FUNCTION_BLOCK "GCS7_M_DPScaleMWBL_MWBS"	// FB 61
TITLE = Scale MWBL/MWBS
//  
//COPYRIGHT:    (C) 2001  BUHLER AG, CH-9240 UZWIL, SWITZERLAND
//
//PRODUCT:      GCS7
//
//TITLE:        FB 61 Machine Control:Scale MWBL/MWBS
//              (with FB40) 
//-------------------------------------------------------------------------
//
//IDENT:        AUTHOR:             DEPT:                       DATE:
//
//FB61.2.1      A. Egli             CT3                         17-Mai-2004
//              Scale.InDisableDischargeDUMP moved to last netzwerk
//              Scale not interlocked with InDisableAirlock 
//FB61.2.0      A. Egli             CT3                         17-Jun-2002
//              New Release with one block 
//FB61.1.0      A. Egli             CT3                         23-Aug-2001
//              Make new Version FB62.5.1 with DP Scales
//
//-------------------------------------------------------------------------
//
//PURPOSE:      MANUAL : see [LL.MWBxxMAN]
//
//RESTRICTIONS: S7
//              ACCU2: Pointer to dynamic datas of the machine
//              ACCU1: Pointer to parameter datas of the machine
//              >=FB26.1.0 
//
//-------------------------------------------------------------------------
//
//
AUTHOR : EA
FAMILY : GCS7LL
NAME : Ma_MWBL
VERSION : 2.1
VAR
  Ma : UDT 20610;
  Airlock : FB 12;	//Element
  LLOutlet : FB 14;	//Element
  HLInlet : FB 14;	//Element
  Scale : FB 40;	//Element
END_VAR
VAR_TEMP
  tmpFaultStop : BOOL ;
  tmpFaultSum : BOOL ;
  tmpNext : BOOL ;
  tmpNext2 : BOOL ;
  tmpEnable : BOOL ;
  tmpEmpty : BOOL ;
  tmpDisableAirlock : BOOL ;
  tmpLenDyn : INT ;
  tmpStoreAR2 : DINT ;
END_VAR
BEGIN
NETWORK
TITLE =
      L     12;
      T     #tmpLenDyn;
NETWORK
TITLE = PC Control
      NOP   0;
//=== Test Object number =====================
      L     "SYS_DirectCtrlDB".PC.ObjectNo;	//PCControl.ObjectNo
      L     #Ma.Par.ParObjectNo;	//Input ObjectNo
      <>I;
      JC    aEnd;
//=== Test OType      ========================
      L     2061;	//Input object type
      L     "SYS_DirectCtrlDB".PC.ObjectType;	//PCControl.ObjectType
      <>I;
      JC    aEnd;
//=== Test Handshake =========================
      A     "SYS_DirectCtrlDB".PC.Hsk.FExamine;	// Handshake.FExamine
      JC    aExa;
      A     "SYS_DirectCtrlDB".PC.Hsk.FDefineCmd;	// Handshake.FDefineCmd
      O     "SYS_DirectCtrlDB".PC.Hsk.FDefinePara;	// Handshake.FDefinePara
      JC    aCmd;
aIni: L     2;	// FcInit
      UC    "SYS_DirectCtrl";
      JU    aEnd;
// Write new commands from PC to Interface of group 
aCmd: A     "SYS_DirectCtrlDB".PC.Cmd1[8];	//Cmd1[8]=CmdOff
      S     #Ma.CmdOff;
      A     "SYS_DirectCtrlDB".PC.Cmd1[9];	//Cmd1[9]=CmdOn
      S     #Ma.CmdOn;
      A     "SYS_DirectCtrlDB".PC.Cmd1[10];	//Cmd1[10]=CmdNext
      S     #Ma.CmdNext;
      A     "SYS_DirectCtrlDB".PC.Cmd1[11];	//Cmd1[11]=CmdFaultReset
      S     #Ma.CmdFaultReset;
      A     "SYS_DirectCtrlDB".PC.Cmd1[13];	//Cmd1[13]=CmdManualOn
      S     #Ma.InManual;
      A     "SYS_DirectCtrlDB".PC.Cmd2[13];	//Cmd1[13]=CmdManualOff
      R     #Ma.InManual;
//[4.0]   U     PCControl.PC.Cmd1[1]; //Cmd1[1]=CmdEmptyingOn
//[4.0]   S     #Ma.InRestdischarge;
//[4.0]   U     PCControl.PC.Cmd2[1]; //Cmd2[1]=CmdEmptyingOff
//[4.0]   R     #Ma.InRestdischarge; 
      A     "SYS_DirectCtrlDB".PC.Cmd1[2];	//Cmd1[2]=CmdDisableAirlock
      S     #Ma.InDisableAirlock;
      A     "SYS_DirectCtrlDB".PC.Cmd2[2];	//Cmd2[2]=CmdEnableAirlock
      R     #Ma.InDisableAirlock;
      A     "SYS_DirectCtrlDB".PC.Cmd1[7];	//Cmd2[2]=CmdEmptying
      S     #Ma.InOutEmptyingHopperScale;
      A     "SYS_DirectCtrlDB".PC.Cmd1[4];	//Cmd1[4]=CmdNewValue
      S     #Ma.CmdNewValue;
      A     "SYS_DirectCtrlDB".PC.Cmd1[5];	//Cmd1[5]=CmdNewJob
      S     #Ma.CmdNewJob;
      AN    "SYS_DirectCtrlDB".PC.Hsk.FDefinePara;	// Handshake.FDefinePara
      JC    aIni;
      JU    aIni;
aExa: TAR2;	// Address Dynamic data
      T     "SYS_DirectCtrlDB".GC.InDynAddr;	// -->PCControl.GC.InDynAddr
      L     #tmpLenDyn;	// Length Dynamic data
      T     "SYS_DirectCtrlDB".GC.InDynLen;	// -->PCControl.GC.InDynLen
      L     0;
      T     "SYS_DirectCtrlDB".GC.InParaAddr;	// -->PCControl.GC.InParaAddr
      T     "SYS_DirectCtrlDB".GC.InParaLen;	// -->PCControl.GC.InParaLen
      L     1;	// Code FcExamine
      UC    "SYS_DirectCtrl";
      L     10;	//Revision
      T     "SYS_DirectCtrlDB".GC.Revision;
aEnd: NOP   0;
NETWORK
TITLE = Interlocking
      NOP   0;
//===Global Group Orders===
      A     "GCS7_Gr_OutManualOn";	//Gr.OutManualOn
      S     #Ma.InManual;
      A     "GCS7_Gr_OutManualOff";	//Gr.OutManualOff
      R     #Ma.InManual;
      A     #Ma.InManual;
      S     "GCS7_Gr_InManual";	//Gr.InManual
      A     #Ma.CmdNext;
      AN    #Ma.InManual;
      O     #Ma.CmdOn;
      =     #tmpNext;
      A     #Ma.InManual;
      ON    #Ma.InLocal;
      A     #Ma.InEnable;
      AN    #Ma.CmdOff;
      =     #tmpEnable;
// Continue after Empyting
      A     #Ma.CmdNewJob;
      O     #Ma.CmdOn;
      ON    #tmpEnable;
      R     #Ma.InOutEmptyingHopperScale;	//[4.0]
//---- Low level 
      A     #HLInlet.StFalse;
      O     #HLInlet.StFault;
      O     #HLInlet.StCtoTrue;
      =     #Ma.OutEmptyInlet;
      A     #Ma.OutEmptyInlet;
      AN    #Ma.InOutEmptyingHopperScale;	//[4.0]
      A     #Ma.Par.ParWithHLInlet;
      =     #tmpEmpty;
      A     #LLOutlet.StFalse;
      O     #LLOutlet.StCtoTrue;
      =     #Ma.OutEmptyOutlet;
//--- Fault----
      O     #HLInlet.StFault;
      O     #LLOutlet.StFault;
      O     #Airlock.StFault;
      O     #Scale.StFault;
      =     #tmpFaultSum;
// 
//--- Interlocking Airlock
      A     #Ma.OutEmptyOutlet;
      AN    #Ma.InOutEmptyingHopperScale;	//[4.0]
      A     #Ma.Par.ParStopAirlockByLL;
      O     #Ma.InDisableAirlock;
      =     #tmpDisableAirlock;
      AN    #tmpDisableAirlock;
      A     #tmpEnable;
      =     #Airlock.InEnableFwd;
//[4.0->] Sequence stop DUMP scale
      AN    #Ma.InManual;
      A     #Ma.InSeqStop;
      =     #Scale.InSeqStopDUMP;	//Emptying scale, but not hopper above scale
      A     #Scale.InSeqStopDUMP;
      AN    #Scale.StDosing;
      AN    #Scale.StStarting;	//[<-4.0]
      =     #Airlock.InSeqStop;
// 
      A     #Ma.StStarted;
      O     #Ma.StEmptying;
      O     #Ma.StEmptied;
      O     #Ma.StWaiting;
      AN    #Ma.InLocal;
      AN    #Ma.InManual;
      O     #tmpNext;
      S     #Airlock.CmdNext;
      =     #tmpNext2;
// 
//--- Interlocking Scale
//[2.1]      UN    #Ma.InDisableAirlock        //[4.0] Stop scale,
//[2.1]      O     #Ma.Par.ParWithLLOutlet     //[4.0]  if no HLOutlet is used
      AN    #Airlock.StFault;
      A(;
      ON    #Airlock.StStopped;
      ON    #Ma.Par.ParWithAirlock;
      ON    #Ma.InSeqStop;
      );
      A     #tmpEnable;
      =     #Scale.InEnable;
//[2.1] Scale.InDisableDischargeDUMP moved to last netzwerk
// 
      A     #Ma.InOutEmptyingHopperScale;	//[4.0]
      AN    #Scale.InManual;
      O;
      A     #Scale.InManual;
      A     #Scale.InOutRestdischargeBin;	//[4.0]
      =     #Scale.InOutRestdischargeBin;	//[4.0]
// 
      AN    #Airlock.InEnableFwd;
      O     #Airlock.StStartedFwd;
      O     #tmpDisableAirlock;
      ON    #Ma.Par.ParWithAirlock;
      A     #tmpNext2;
      S     #Scale.CmdNext;
      A     #Ma.CmdOff;
      S     #Scale.CmdOff;
//New job 
      A     #Ma.CmdNewJob;
      S     #Scale.CmdNewJob;
      A     #Ma.CmdNewValue;
      S     #Scale.CmdNewValue;
// 
//--- Local mode --
      A     #Ma.InLocal;
      AN    #Ma.InManual;
      =     #Scale.InLocal;
      =     #Airlock.InLocal;
      =     #HLInlet.InLocal;
      A     #Scale.InLocal;	//[4.0]
      O     #Ma.Par.ParHLOutletLocal;	//[4.0]
      =     #LLOutlet.InLocal;
//--- Monitoring -------------
      A     #Airlock.StStartedFwd;
      ON    #Ma.Par.ParWithAirlock;
      O     #Scale.StDosing;
      =     #LLOutlet.InMonFalse;
//--- Fault Reset -------------
      A     #Ma.CmdFaultReset;
      S     #Scale.CmdFaultReset;
      S     #Airlock.CmdFaultReset;
      S     #HLInlet.CmdFaultReset;
      S     #LLOutlet.CmdFaultReset;
//--- Stop Point -------------
      A     #Scale.OutStopPoint;
      =     #Ma.OutStopPoint;
NETWORK
TITLE = Call Scale
      CALL  #Scale;	// Call Scale
NETWORK
TITLE = Call Motor: Airlock
      AN    #Ma.Par.ParWithAirlock;
      JC    el3;
      CALL  #Airlock;
NETWORK
TITLE = Call Digital Input: HLOutlet
el3:  AN    #Ma.Par.ParWithLLOutlet;
      JC    el4;
      CALL  #LLOutlet;
NETWORK
TITLE = Call Digital Input: LLInlet
el4:  AN    #Ma.Par.ParWithHLInlet;
      JC    StJ0;
      CALL  #HLInlet;
NETWORK
TITLE = Jump to actual state
StJ0: A     #Ma.StStopped;
      JC    S0;	// ===> State
      A     #Ma.StStarted;
      JC    S2;	// ===> State
      A     #Ma.StStarting;
      JC    S1;	// ===> State
      A     #Ma.StStopping;
      JC    S3;	// ===> State
      A     #Ma.StFault;
      JC    S4;	// ===> State
      A     #Ma.StWaiting;
      JC    S5;	// ===> State
      A     #Ma.StEmptying;
      JC    S6;	// ===> State
      A     #Ma.StEmptied;
      JC    S7;	// ===> State
NETWORK
TITLE = Stopped
xxS0: S     #Ma.StStopped;	// any Transition ===> Initialisation
//=== Logic
// Condition for StFault
S0:   A     #tmpFaultSum;
      R     #Ma.StStopped;
      JC    xxS4;	//--> ST_FAULT:
// Condition for StStarting
      AN    #Airlock.StStopped;
      A     #Ma.Par.ParWithAirlock;
      ON    #Scale.StStopped;
      R     #Ma.StStopped;
      JC    xxS1;	//--> StStarting
// Condition for StWaiting
      A     #tmpNext;
      A     #tmpEnable;
      A     #tmpEmpty;
      R     #Ma.StStopped;
      JC    xxS5;	//--> StWaiting
      JU    OUT;
NETWORK
TITLE = StStarting
xxS1: S     #Ma.StStarting;	//any Transition 
//=== Logic
// Condition for StFault
S1:   A     #tmpFaultSum;
      R     #Ma.StStarting;
      JC    xxS4;	//--> StFault
// Condition for StStarted
      A     #Scale.StDosing;
      R     #Ma.StStarting;
      JC    xxS2;	//-->StStarted
// Condition for StEmptying
      A     #Scale.StEmptying;
      O     #Scale.StEmptied;
      R     #Ma.StStarting;
      JC    xxS6;	//--> StEmptying
// Condition for StStopping
      AN    #Airlock.StStartedFwd;
      O     #Airlock.InSeqStop;
      AN    #Airlock.StStarting;
      AN    #Scale.StStarting;
      AN    #Scale.InEnable;
      R     #Ma.StStarting;
      JC    xxS3;	//-->StStopping
      JU    OUT;
NETWORK
TITLE = StStarted
xxS2: S     #Ma.StStarted;	//any Transition 
//=== Logic
// Condition for StFault
S2:   A     #tmpFaultSum;
      R     #Ma.StStarted;
      JC    xxS4;	//--> StFault
// Condition for StEmptying
      A     #Scale.StEmptying;
      O     #Scale.StEmptied;
      R     #Ma.StStarted;
      JC    xxS6;	//-->StEmptying
// Condition for StWaiting
//[4.0]   U     #tmpEmpty;     
      AN    #Ma.OutEmptyOutlet;
      ON    #Ma.Par.ParWithLLOutlet;	//[4.0]
      AN    #Ma.InOutEmptyingHopperScale;	//[4.0]
      A(;	//[5.0][PE]
      AN    #Scale.StDosing;
      O     #Scale.InDisableDischargeDUMP;	//[5.0][PE]
      );	//[5.0][PE]
      R     #Ma.StStarted;
      JC    xxS5;	//-->StWaiting
// Condition for StStopping
      AN    #Scale.StDosing;
      R     #Ma.StStarted;
      JC    xxS3;	//-->StStopping
      JU    OUT;
NETWORK
TITLE = Stopping
xxS3: S     #Ma.StStopping;	//any Transition 
//=== Logic
// Condition for StFault
S3:   A     #tmpFaultSum;
      R     #Ma.StStopping;
      JC    xxS4;	//--> StFault
// Condition for StStopped
      A     #Airlock.StStopped;
      ON    #Ma.Par.ParWithAirlock;
      A     #Scale.StStopped;
      R     #Ma.StStopping;
      JC    xxS0;	//-->StStopped
// Condition for StStarting
      A     #Airlock.StStartedFwd;
      AN    #Airlock.InSeqStop;
      O     #Scale.StDosing;
      O     #Scale.InEnable;
      R     #Ma.StStopping;
      JC    xxS1;	//-->StStarting
      JU    OUT;
NETWORK
TITLE = Fault
xxS4: S     #Ma.StFault;	//any Transition 
      JU    OUT;
//=== Logic
S4:   A     #tmpFaultSum;
      JC    OUT;
//---- Transition --
      R     #Ma.StFault;
      JU    xxS3;	//-->StStopping 
NETWORK
TITLE = StWaiting
xxS5: S     #Ma.StWaiting;	//any Transition 
      JU    OUT;
//=== Logic
// Condition for StFault
S5:   A     #tmpFaultSum;
      R     #Ma.StWaiting;
      JC    xxS4;	//--> StFault
// Condition for StDosing
      A     #Scale.StDosing;
      AN    #Scale.InDisableDischargeDUMP;	//[5.0][PE]
      R     #Ma.StWaiting;
      JC    xxS2;	//-->StDosing
// Condition for StEmptying             // [4.1]
      A     #Scale.StEmptying;	// [4.1]
      A     #LLOutlet.StFalse;	// [4.1]
      R     #Ma.StWaiting;	// [4.1]
      JC    xxS6;	//-->StEmptying // [4.1]
// Condition for StEmptied              // [4.1]
      A     #Scale.StEmptied;	// [4.1]
      A     #LLOutlet.StFalse;	// [4.1]
      R     #Ma.StWaiting;	// [4.1]
      JC    xxS7;	//-->StEmptied  // [4.1]
// Condition for StStopping
      AN    #tmpEnable;
      R     #Ma.StWaiting;
      JC    xxS0;	//-->StStopping
      JU    OUT;
NETWORK
TITLE = StEmptying
xxS6: S     #Ma.StEmptying;	//any Transition 
      JU    OUT;
//=== Logic
// Condition for StFault
S6:   A     #tmpFaultSum;
      R     #Ma.StEmptying;
      JC    xxS4;	//--> StFault
// Condition for StEmptied
      A     #Scale.StEmptied;
      R     #Ma.StEmptying;
      JC    xxS7;	//-->StEmptied
// Condition for StStopping
      AN    #Scale.StEmptying;
      R     #Ma.StEmptying;
      JC    xxS3;	//-->StStopping
      JU    OUT;
NETWORK
TITLE = StEmptied
xxS7: S     #Ma.StEmptied;	//any Transition 
      JU    OUT;
//=== Logic
// Condition for StFault
S7:   A     #tmpFaultSum;
      R     #Ma.StEmptied;
      JC    xxS4;	//--> StFault
// Condition for StStarted
      A     #Scale.StDosing;
      R     #Ma.StEmptied;
      JC    xxS2;	//-->StStarted
// Condition for StStopping
      AN    #Scale.StEmptied;
      AN    #Scale.StStarting;
      R     #Ma.StEmptied;
      JC    xxS3;	//-->StStopping
      JU    OUT;
NETWORK
TITLE = State Code
// State     StCode
// ----------------------
// StFault32
// StStopped    1
// StStarting   2
// StWaiting    3
// StStarted    4
// StStopping    7
// StEmptying     9
// StEmptied        10
OUT:  A     #Ma.StStopped;
      L     1;	//Code=StStopped
      JC    Code;
      A     #Ma.StStarted;
      L     4;	//Code=StStarted
      JC    Code;
      A     #Ma.StWaiting;
      L     3;	//Code=StWaiting
      JC    Code;
      A     #Ma.StStarting;
      L     2;	//Code=StStarting
      JC    Code;
      A     #Ma.StStopping;
      L     7;	//Code=StStopping
      JC    Code;
      A     #Ma.StEmptying;
      L     9;	//Code=StEmptying
      JC    Code;
      A     #Ma.StEmptied;
      L     10;	//Code=StEmptied
      JC    Code;
      L     32;	//Code=StFault 
Code: L     #Ma.StCode;	// Old state code
      TAK;
      T     #Ma.StCode;	// Save state code
      <>I;
      L     3;
      CC    "SYS_CBitCtrl";	//Set change bit
NETWORK
TITLE = Global End
      CLR;	//---Clear all commands
      =     #Ma.CmdOn;
      =     #Ma.CmdOff;
      =     #Ma.CmdNext;
      =     #Ma.CmdFaultReset;
      =     #Ma.CmdNewValue;
      =     #Ma.CmdNewJob;
//[2.1] Scale.InDisableDischargeDUMP moved to last netzwerk
      A     #Ma.InDisableAirlock;	//[2.1] Stop scale,
      AN    #Ma.Par.ParWithLLOutlet;	//[2.1]  if no HLOutlet is used
      O(;
      A     #LLOutlet.StFault;	//[5.0][PE]
      O     #LLOutlet.StTrue;	//[5.0][PE]
      O     #LLOutlet.StCtoFalse;	//[5.0][PE]
      A     #Ma.Par.ParWithLLOutlet;	//[2.1]
      );	//[2.1]
      =     #Scale.InDisableDischargeDUMP;	//[5.0][PE]
END_FUNCTION_BLOCK

FUNCTION_BLOCK "GCS7_M_DriveCurrent"	// FB 62
TITLE = Motor with bypass flap
//  
//COPYRIGHT:    (C) 1997  BUHLER AG, CH-9240 UZWIL,  SWITZERLAND
//
//PRODUCT:      GCS7
//
//TITLE:        FB 62 Machine Control:Drive with Current
//-------------------------------------------------------------------------
//
//IDENT:        AUTHOR:             DEPT:                       DATE:
//
//FB62.1.0      A.Egli              CT3                         5-Jul-2004
//              1st Release in S7
//
//-------------------------------------------------------------------------
//
//PURPOSE:      MANUAL : see [LL.DRCUxxMAN]
//
//RESTRICTIONS: S7
//
//-------------------------------------------------------------------------
//
AUTHOR : EA
FAMILY : GCS7LL
NAME : DRCU
VERSION : 1.0
VAR
  Ma : UDT 20620;
  Mon1 : FB 14;	//Element
  Current : FB 19;	//Element [4.0]
  Motor : FB 12;	//Element
  Release : FB 11;	//Element
END_VAR
VAR_TEMP
  tmpFaultSum : BOOL ;
  tmpLocal : BOOL ;
  tmpEnable : BOOL ;
  tmpStartReq : BOOL ;
  tmpLenDyn : INT ;
  tmpEnableRelease : BOOL ;
END_VAR
BEGIN
NETWORK
TITLE =
      L     22;
      T     #tmpLenDyn;
NETWORK
TITLE = PC Control
//=== Test Object number =====================
      L     "SYS_DirectCtrlDB".PC.ObjectNo;	//PCControl.ObjectNo
      L     #Ma.Par.ParObjectNo;	//Input ObjectNo
      <>I;
      JC    aEnd;
//=== Test OType      ========================
      L     2062;	//Input object type
      L     "SYS_DirectCtrlDB".PC.ObjectType;	//PCControl.ObjectType
      <>I;
      JC    aEnd;
//=== Test Handshake =========================
      A     "SYS_DirectCtrlDB".PC.Hsk.FExamine;	// Handshake.FExamine
      JC    aExa;
      A     "SYS_DirectCtrlDB".PC.Hsk.FDefineCmd;	// Handshake.FDefineCmd
      JC    aCmd;
      A     "SYS_DirectCtrlDB".PC.Hsk.FDefinePara;	// Handshake.FDefinePara
      JC    pPar;
aIni: L     2;	// FcInit
      UC    "SYS_DirectCtrl";
      JU    aEnd;
// Write parameter 
pPar: LAR1  P#DBX 58.0;
      L     P#6.0;
      +AR1;
      L     DBW [AR1,P#4.0];
      T     #Ma.Par.ParClearingTime;
// Write new commands from PC to Interface of group 
aCmd: A     "SYS_DirectCtrlDB".PC.Cmd1[8];	//Cmd1[8]=CmdOff
      S     #Ma.CmdOff;
      A     "SYS_DirectCtrlDB".PC.Cmd1[9];	//Cmd1[9]=CmdOn
      S     #Ma.CmdOn;
      A     "SYS_DirectCtrlDB".PC.Cmd1[10];	//Cmd1[10]=CmdNext
      S     #Ma.CmdNext;
      A     "SYS_DirectCtrlDB".PC.Cmd1[11];	//Cmd1[11]=CmdFaultReset
      S     #Ma.CmdFaultReset;
      A     "SYS_DirectCtrlDB".PC.Cmd1[13];	//Cmd1[13]=CmdManualOn
      S     #Ma.InManual;
      A     "SYS_DirectCtrlDB".PC.Cmd2[13];	//Cmd2[13]=CmdManualOff
      R     #Ma.InManual;
      R     #Motor.InManual;
      R     #Release.InManual;
      JU    aIni;
aExa: TAR2;	// Address dynamic data
      T     "SYS_DirectCtrlDB".GC.InDynAddr;	// -->PCControl.GC.InDynAddr
      L     #tmpLenDyn;	// Length Dynamic data
      T     "SYS_DirectCtrlDB".GC.InDynLen;	// -->PCControl.GC.InDynLen
      L     0;
      T     "SYS_DirectCtrlDB".GC.InParaAddr;	// -->PCControl.GC.InParaAddr
      T     "SYS_DirectCtrlDB".GC.InParaLen;	// -->PCControl.GC.InParaLen
      L     1;	// Code FcExamine
      UC    "SYS_DirectCtrl";
      L     10;	//Revision
      T     "SYS_DirectCtrlDB".GC.Revision;
aEnd: NOP   0;
NETWORK
TITLE = Interlocking
//===Global Group Orders===
      A     "GCS7_Gr_OutManualOn";	//Gr.OutManualOn
      S     #Ma.InManual;
      A     "GCS7_Gr_OutManualOff";	//Gr.OutManualOff
      R     #Ma.InManual;
      A     #Ma.InManual;
      S     "GCS7_Gr_InManual";	//Gr.InManual
      A     #Ma.InLocal;
      AN    #Ma.InManual;
      =     #tmpLocal;
//--- Fault----
      A     #Current.OutFaulted;
      A     #Ma.InMonFault;
      O     #Mon1.StFault;
      O     #Motor.StFault;
      O     #Release.StFault;
      =     #tmpFaultSum;
//---Enable----
      AN    #Ma.CmdOff;
      A     #Ma.InEnable;
      =     #tmpEnable;
//--- Local mode --
      A     #tmpLocal;
      =     #Motor.InLocal;
      =     #Mon1.InLocal;
      =     #Release.InLocal;
      =     #Current.InLocal;
//--- Fault Reset -------------
      A     #Ma.CmdFaultReset;
      S     #Mon1.CmdFaultReset;
      S     #Motor.CmdFaultReset;
      S     #Release.CmdFaultReset;
      S     #Current.CmdFaultReset;
NETWORK
TITLE = Loaded
      A     #Ma.InFeeding;
      O     #Current.OutL;
      S     #Ma.OutLoaded;
      S     #Ma.OutMonitoring;
      AN    #Motor.StStartedFwd;
      R     #Ma.OutMonitoring;
NETWORK
TITLE = Interlocking Motor
//InEnableXxx
      AN    #Current.OutFaulted;
      ON    #Ma.InMonFault;
      AN    #Mon1.StFault;
      A     #Ma.InEnable;
      A(;
      A     #Ma.OutLoaded;
      ON    #Ma.InClearing;
      );
      =     #Motor.InEnableFwd;
//CmdNext
      AN    #Ma.InManual;
      A     #Ma.CmdNext;
      A     #Motor.InEnableFwd;
      O;
      A     #Ma.InManual;
      A     #Ma.CmdOn;
      S     #Motor.CmdNext;
//CmdSeqStop
      A     #Ma.InSeqStop;
      =     #Motor.InSeqStop;
NETWORK
TITLE = Interlocking Element Release
//--------------
      A     #Motor.StStartedFwd;
      A     #Ma.OutLoaded;
      A     #Ma.InReleaseOutput;
      =     #tmpEnableRelease;
      JC    erJ1;
      L     #Ma.Par.ParDelayRelease;
      T     #Ma.Par.OutDelayDosing;
      JU    erJ2;
erJ1: AN    "GCS7_Gr_OutTick200ms";
      O     #Release.InEnable;
      JC    erJ2;
      L     #Ma.Par.OutDelayDosing;
      +     -2;
      T     #Ma.Par.OutDelayDosing;
erJ2: L     #Ma.Par.OutDelayDosing;
      L     0;
      <=I;
      A     #tmpEnableRelease;
      =     #Release.InEnable;
      SET;
      S     #Release.CmdNext;
NETWORK
TITLE = Monitoring Element Mon1
      A     #Motor.StStartedFwd;
      O     #Motor.StStartedRev;
      =     #Mon1.InMonTrue;
      CLR;
      =     #Mon1.InMonFalse;
NETWORK
TITLE = Monitoring Element Current
//Set Parameter
      L     #Ma.Par.ParCurrentNom;
      T     #Current.Par.ParLimitL;
      L     100;
      L     #Ma.Par.ParLimitMin;
      -D;
      DTR;
      L     #Ma.Par.ParCurrentNom;
      DTR;
      *R;
      L     1.000000e+02;
      /R;
      RND;
      T     #Current.Par.ParLimitLL;
      L     #Ma.Par.ParLimitMax;
      L     100;
      +I;
      DTR;
      L     #Ma.Par.ParCurrentNom;
      DTR;
      *R;
      L     1.000000e+02;
      /R;
      RND;
      T     #Current.Par.ParLimitHH;
      T     #Current.Par.ParLimitH;
      SET;
      R     #Current.Par.ParLimitsPc;
      AN    #Ma.InMonFault;
      =     #Current.Par.ParWarningLL;
      =     #Current.Par.ParWarningL;
      =     #Current.Par.ParWarningH;
      =     #Current.Par.ParWarningHH;
//Monitoring
      A     #Ma.OutMonitoring;
      =     #Current.InMonLL;
      =     #Current.InMonL;
      CLR;
      =     #Current.InMonMid;
      A     #Ma.OutMonitoring;
      =     #Current.InMonH;
      =     #Current.InMonHH;
      A     #Current.OutWarning;
      O     #Current.OutFaulted;
      A     #Motor.StStartedFwd;
      AN    #Ma.InMonFault;
      =     #Ma.OutWarning;
NETWORK
TITLE = Call Digital Input: Monitor 
      AN    #Ma.Par.ParWithMon1;
      JC    Moto;
      CALL  #Mon1;
NETWORK
TITLE = Call Motor
Moto: CALL  #Motor;
NETWORK
TITLE = Call Release
      AN    #Ma.Par.ParWithRelease;
      JC    Curr;
      CALL  #Release;
NETWORK
TITLE = Call Current
Curr: CALL  #Current;
NETWORK
TITLE = Jump to actual state
      A     #Ma.StStopped;
      JC    S0;	// ===> State
      A     #Ma.StStarted;
      JC    S2;	// ===> State
      A     #Ma.StStarting;
      JC    S1;	// ===> State
      A     #Ma.StStopping;
      JC    S3;	// ===> State
      A     #Ma.StClearing;
      JC    S5;	// ===> State
      A     #Ma.StDosing;
      JC    S6;	// ===> State
      A     #Ma.StFault;
      JC    S4;	// ===> State
NETWORK
TITLE = Stopped
xxS0: S     #Ma.StStopped;
S0:   A     #tmpFaultSum;
      R     #Ma.StStopped;
      JC    xxS4;	//--> StFault
      AN    #Motor.StStopped;
      R     #Ma.StStopped;
      JC    xxS1;	//--> StStarting
      JU    OUT;
NETWORK
TITLE = Starting
xxS1: S     #Ma.StStarting;
S1:   A     #tmpFaultSum;
      R     #Ma.StStarting;
      JC    xxS4;	//--> StFault
// Condition for StStopping
      A     #Motor.StStopped;
      O     #Motor.StStopping;
      R     #Ma.StStarting;
      JC    xxS3;	//--> StStopping
// Condition for StStarted
      A(;
      O     #Motor.StStartedFwd;
      O     #Motor.StStartedRev;
      );
      R     #Ma.StStarting;
      JC    xxS2;	//--> StStarted
      JU    OUT;
NETWORK
TITLE = Started
xxS2: S     #Ma.StStarted;
S2:   A     #tmpFaultSum;
      R     #Ma.StStarted;
      JC    xxS4;	//--> StFault
// Condition for StStopping
      AN    #Motor.StStartedRev;
      AN    #Motor.StStartedFwd;
      R     #Ma.StStarted;
      JC    xxS3;	//--> StStopping
// Condition for StEnabled
      A     #Release.StStarted;
      R     #Ma.StStarted;
      JC    xxS6;	//--> StReleased
// Condition for StClearing
      A     #Ma.InClearing;
      R     #Ma.StStarted;
      JC    xxS5;	//--> StClearing
      JU    OUT;
NETWORK
TITLE = StClearing
//any Transition 
xxS5: S     #Ma.StClearing;
      L     #Ma.Par.ParClearingTime;
      T     #Ma.Par.OutClearingTime;
//=== Logic
// Condition for StFault
S5:   A     #tmpFaultSum;
      R     #Ma.StClearing;
      JC    xxS4;	//--> StFault
// Condition for StStarted
      AN    #Motor.StStartedFwd;
      AN    #Motor.StStartedRev;
      ON    #Ma.InClearing;
      R     #Ma.StClearing;
      JC    xxS2;	//--> StStarted
// Condition for StBypassed
      L     0;
      L     #Ma.Par.OutClearingTime;
      >=I;
      R     #Ma.OutLoaded;
      JC    xxS6;	//--> StBypassed
//Clearing Time
      ON    "GCS7_Gr_OutTick500ms";	//Gr.OutTick500ms
      JC    OUT;
      L     #Ma.Par.OutClearingTime;
      +     -5;
      T     #Ma.Par.OutClearingTime;
      JU    OUT;
NETWORK
TITLE = StDosing
//any Transition 
xxS6: S     #Ma.StDosing;
//=== Logic
// Condition for StFault
S6:   A     #tmpFaultSum;
      R     #Ma.StDosing;
      JC    xxS4;	//--> StFault
// Condition for StStarted
      AN    #Release.StStarted;
      R     #Ma.StDosing;
      JC    xxS2;	//--> StStarted
// Condition for StStopping
      AN    #Motor.StStartedFwd;
      AN    #Motor.StStartedRev;
      R     #Ma.StDosing;
      JC    xxS3;	//--> StStopping
// Condition for StClearing
      A     #Ma.InClearing;
      R     #Ma.StDosing;
      JC    xxS5;	//--> StClearing
      JU    OUT;
NETWORK
TITLE = Stopping
xxS3: S     #Ma.StStopping;
S3:   A     #tmpFaultSum;
      R     #Ma.StStopping;
      JC    xxS4;	//--> StFault
// Condition for StStopped
      A     #Motor.StStopped;
      R     #Ma.StStopping;
      JC    xxS0;	//--> StStopped
// Condition for StStarting
      AN    #Motor.StStopping;
      R     #Ma.StStopping;
      JC    xxS1;	//--> StStarting
      JU    OUT;
NETWORK
TITLE = Fault
xxS4: S     #Ma.StFault;
S4:   AN    #tmpFaultSum;
      R     #Ma.StFault;
      JC    xxS3;	//--> StStopping
      JU    OUT;
NETWORK
TITLE = Global End
OUT:  CLR;	//---Clear all commands
      =     #Ma.CmdOn;
      =     #Ma.CmdOff;
      =     #Ma.CmdNext;
      =     #Ma.CmdFaultReset;
NETWORK
TITLE = State Code
// 1=StStopped    11=StStopped.Warning
// 2=StStarting   12=StStarting.Warning
// 3=StStarted    13=StStarted.Warning
// 4=StDosing     15=StDosing.Warning
// 6=StClearing   16=StClearing.Warning
// 7=StStopping   17=StStopping.Warning
//32=StFault
      L     32;	// StCode=Fault
      A     #Ma.StFault;
      JC    Code;
      L     1;	// StCode=Stopped
      A     #Ma.StStopped;
      JC    Cod1;
      L     2;	// StCode=Starting
      A     #Ma.StStarting;
      JC    Cod1;
      L     3;	// StCode=Started
      A     #Ma.StStarted;
      JC    Cod1;
      L     6;	// StCode=Clearing
      A     #Ma.StClearing;
      JC    Cod1;
      L     4;	// StCode=Dosing
      A     #Ma.StDosing;
      JC    Cod1;
      L     7;	// StCode=Stopping
Cod1: AN    #Ma.OutWarning;
      JC    Code;
      +     10;
Code: L     #Ma.StCode;	// Old state code
      TAK;
      T     #Ma.StCode;	// Save state code
      <>I;
      L     3;
      CC    "SYS_CBitCtrl";	//Set change bit
END_FUNCTION_BLOCK

FUNCTION_BLOCK "GCS7_M_DFCA"	// FB 63
TITLE = Machine DFCA, DFCB, DFBB Control
//
//COPYRIGHT:    (C) 2001  BUHLER AG, CH-9240 UZWIL, SWITZERLAND
//
//PRODUCT:      GCS7
//
//TITLE:        Machine DFCA, DFCB, DFBB Control
//              (GCPROVB Revision 11)
//-------------------------------------------------------------------------
//
//IDENT:        AUTHOR:             DEPT:                       DATE:
//
//FB63.5.0      A. Egli             CT3                         26-Oct-2004
//              FB73.5.0 with B106 
//FB63.4.0      A. Egli             CT3                         08-Dez-2003
//              FB73 with A202 
//FB63.3.0      A. Egli             CT3                         17-Jun-2002
//              DFCB, DFBB 
//FB63.2.0      A. Egli             CT3                         17-Jun-2002
//              New Release with one block 
//FB63.1.1      Ph. Engler          MU664                       31-Oct-2001
//              No Press.cmdStart if InSuspend
//FB63.1.0      A. Egli             CT3                         17-Jul-2001
//              1st Release in S7
//
//-------------------------------------------------------------------------
//
//PURPOSE:      MANUAL : see [MxxMAN]
//
//RESTRICTIONS: 
//
//-------------------------------------------------------------------------
//
AUTHOR : EA
FAMILY : GCS7LL
NAME : MA_DFCA
VERSION : 5.0
VAR
  Ma : UDT 20630;
  ElRemote : FB 14;	//Input from DFCA: (DP or Dig. Input) : Freigabe Fernbetrieb
  ElRunning : FB 14;	//Input from DFCA: (DP or Dig. Input) : Betrieb, Ganze Maschine läuft
  ElSumFault : FB 14;	//Input from DFCA: (DP or Dig. Input) : Sammelalarm
  ElFireAlarm : FB 14;	//Input from DFCA: (Dig. Input      ) : Branschutzalarm
  ElPressStart : FB 11;	//Output to DFCA : (DP or Dig. Output): Start an Presse
  ElDischargerRunning : FB 11;	//*O Output to DFCA : (DP or Dig. Output): Abtransport in Betrieb
  ElDPFault : FB 14;	//                    (Internal signal  ): DP Communication fault
  DFxx : FB 73;	//Communication modul
END_VAR
VAR_TEMP
  tmpFaultStop : BOOL ;
  tmpFaultSum : BOOL ;
  tmpLocal : BOOL ;
  tmpEnable : BOOL ;
  tmpLenDyn : INT ;
END_VAR
BEGIN
NETWORK
TITLE =
      L     20;
      T     #tmpLenDyn;
NETWORK
TITLE = Call Communication DFCA
      CALL  #DFxx (
           IOByteNr                 := #Ma.Par.ParIOByteNr);
NETWORK
TITLE = PC Control
//=== Test Object number =====================
      L     "SYS_DirectCtrlDB".PC.ObjectNo;	//PCControl.ObjectNo
      L     #Ma.Par.ParObjectNo;	//Input ObjectNo
      <>I;
      JC    aEnd;
//=== Test OType      ========================
      L     2063;	//Input object type
      L     "SYS_DirectCtrlDB".PC.ObjectType;	//PCControl.ObjectType
      <>I;
      JC    aEnd;
//=== Test Handshake =========================
      A     "SYS_DirectCtrlDB".PC.Hsk.FExamine;	// Handshake.FExamine
      JC    aExa;
      A     "SYS_DirectCtrlDB".PC.Hsk.FDefineCmd;	// Handshake.FDefineCmd
      O     "SYS_DirectCtrlDB".PC.Hsk.FDefinePara;	// Handshake.FDefinePara
      JC    aCmd;
aIni: L     2;	// FcInit
      UC    "SYS_DirectCtrl";
      JU    aEnd;
// Write new commands from PC to Interface of group 
aCmd: A     "SYS_DirectCtrlDB".PC.Cmd1[5];	//Cmd1[8]=CmdNewJob
      S     #Ma.CmdOff;
      A     "SYS_DirectCtrlDB".PC.Cmd1[8];	//Cmd1[8]=CmdOff
      S     #Ma.CmdOff;
      A     "SYS_DirectCtrlDB".PC.Cmd1[9];	//Cmd1[9]=CmdOn
      S     #Ma.CmdOn;
      A     "SYS_DirectCtrlDB".PC.Cmd1[10];	//Cmd1[10]=CmdNext
      S     #Ma.CmdNext;
      A     "SYS_DirectCtrlDB".PC.Cmd1[11];	//Cmd1[11]=CmdFaultReset
      S     #Ma.CmdFaultReset;
      A     "SYS_DirectCtrlDB".PC.Cmd1[13];	//Cmd1[13]=CmdManualOn
      S     #Ma.InManual;
      A     "SYS_DirectCtrlDB".PC.Cmd2[13];	//Cmd2[13]=CmdManualOff
      R     #Ma.InManual;
      A     "SYS_DirectCtrlDB".PC.Cmd1[6];	//Cmd1[6]=InOutCoolerOnMan.On
      S     #Ma.InOutCoolerOnMan;
      A     "SYS_DirectCtrlDB".PC.Cmd2[6];	//Cmd2[6]=Ma.InOutCoolerOnMan.Off
      R     #Ma.InOutCoolerOnMan;
      A     "SYS_DirectCtrlDB".PC.Cmd1[7];	//Cmd1[6]=Ma.InOutHeaterOnMan.On
      S     #Ma.InOutHeaterOnMan;
      A     "SYS_DirectCtrlDB".PC.Cmd2[7];	//Cmd2[6]=Ma.InOutHeaterOnMan.Off
      R     #Ma.InOutHeaterOnMan;
      A     "SYS_DirectCtrlDB".PC.Cmd1[4];	//Cmd1[6]=InOutFanOnMan.On    //[3.0]
      S     #Ma.InOutFanOnMan;
      A     "SYS_DirectCtrlDB".PC.Cmd2[4];	//Cmd2[6]=Ma.InOutFanOnMan.Off   //[3.0]
      R     #Ma.InOutFanOnMan;
      JU    aIni;
aExa: TAR2;	// Address Dynamic datas
      T     "SYS_DirectCtrlDB".GC.InDynAddr;	// -->PCControl.GC.InDynAddr
      L     #tmpLenDyn;	// Length Dynamic datas
      T     "SYS_DirectCtrlDB".GC.InDynLen;	// -->PCControl.GC.InDynLen
      L     0;
      T     "SYS_DirectCtrlDB".GC.InParaAddr;	// -->PCControl.GC.InParaAddr
      T     "SYS_DirectCtrlDB".GC.InParaLen;	// -->PCControl.GC.InParaLen
      L     1;	// Code FcExamine
      UC    "SYS_DirectCtrl";
      L     11;	//Revision
      T     "SYS_DirectCtrlDB".GC.Revision;
aEnd: NOP   0;
NETWORK
TITLE = Interlocking
//===Global Group Orders===
      A     "GCS7_Gr_OutManualOn";	//Gr.OutManualOn
      S     #Ma.InManual;
      A     "GCS7_Gr_OutManualOff";	//Gr.OutManualOff
      R     #Ma.InManual;
      A     #Ma.InManual;
      S     "GCS7_Gr_InManual";	//Gr.InManual
//--- Local mode --
      A     #Ma.InLocal;
      AN    #Ma.InManual;
      =     #tmpLocal;
      A     #tmpLocal;
      =     #ElRemote.InLocal;
      =     #ElRunning.InLocal;
      =     #ElSumFault.InLocal;
      =     #ElFireAlarm.InLocal;
      CLR;
      =     #ElPressStart.InLocal;
      =     #ElDischargerRunning.InLocal;
      A     #tmpLocal;
      ON    #Ma.Par.ParDP;
      =     #ElDPFault.InLocal;
//--- Monitoring
      A     #Ma.InRemoteMode;
      =     #ElRemote.InMonTrue;
      SET;
      =     #ElSumFault.InMonTrue;
      SET;
      =     #ElFireAlarm.InMonTrue;
      A     #Ma.Par.ParDP;
      =     #ElDPFault.InMonTrue;
//--- Fault Reset -------------
      A     #Ma.CmdFaultReset;
      S     #ElRemote.CmdFaultReset;
      S     #ElRunning.CmdFaultReset;
      S     #ElPressStart.CmdFaultReset;
      S     #ElDischargerRunning.CmdFaultReset;
      S     #ElDPFault.CmdFaultReset;
      S     #DFxx.InCommand.CmdFaultResetAll;
      AN    #Ma.CmdFaultReset;
      JC    FRJ1;
      L     #Ma.Par.ParFaultResetTime;
      T     #Ma.Par.OutFaultResetTime;
FRJ1: L     #Ma.Par.OutFaultResetTime;
      L     0;
      <=I;
      ON    "GCS7_Gr_OutTick200ms";
      JC    FRJ2;
      L     #Ma.Par.OutFaultResetTime;
      -I;
      T     #Ma.Par.OutFaultResetTime;
      L     0;
      >I;
      JC    FRJ2;
      S     #ElSumFault.CmdFaultReset;
      S     #ElFireAlarm.CmdFaultReset;
FRJ2: NOP   0;
//=============================================
//ElPressStart: Start/Stop
//=============================================
      A     #Ma.Par.ParManual;
      A     #Ma.InManual;
      O     #Ma.InEnable;
      AN    #Ma.CmdOff;
      =     #tmpEnable;
      A     #Ma.InManual;
      A     #Ma.CmdOn;
      A     #tmpEnable;
      O;
      AN    #Ma.InManual;
      A     #Ma.CmdNext;
      A     #tmpEnable;
      S     #ElPressStart.InEnable;
      S     #ElPressStart.CmdNext;
      AN    #tmpEnable;
      O     #Ma.CmdOff;
      R     #ElPressStart.InEnable;
//=============================================
//ElDischargerRunning
//=============================================
      A     #Ma.InDischargerRunning;
      =     #ElDischargerRunning.InEnable;
      S     #ElDischargerRunning.CmdNext;
NETWORK
TITLE = Commands to DFCA
      A     #ElPressStart.InEnable;
      AN    #Ma.InSuspend;	//[PE]
      =     #DFxx.InCommand.StartPress;
//------------------------------
      AN    #ElPressStart.InEnable;
      =     #DFxx.InCommand.StopPress;
//------------------------------
      A     #Ma.InDischargerRunning;
      =     #DFxx.InCommand.DischargerRunning;
//------------------------------
      A     #Ma.InOutCoolerOnMan;
      =     #DFxx.InCommand.CoolerOnMan;
//------------------------------
      A     #Ma.InOutHeaterOnMan;
      =     #DFxx.InCommand.HeaterOnMan;
//------------------------------
      A     #Ma.InOverrideLLHopper;
      =     #DFxx.InCommand.OverwriteLLHopper;
//------------------------------
      A     #Ma.InSuspend;
      =     #DFxx.InCommand.Suspend;
//------------------------------
      A     #Ma.InOutFanOnMan;	//[3.0]
      =     #DFxx.InCommand.FanOnMan;	//[3.0]
//------------------------------
      A     #Ma.CmdNewJob;
      S     #DFxx.InCommand.CmdResetTotal;
      S     #DFxx.InCommand.CmdResetTotalLiquid1;	//[3.0]
      S     #DFxx.InCommand.CmdResetTotalLiquid2;	//[3.0]
      R     #Ma.CmdNewJob;
//------------------------------
      A     #Ma.CmdResetHorn;
      S     #DFxx.InCommand.CmdResetHorn;
//------------------------------
      CLR;
      S     #DFxx.InCommand.CmdFaultResetSingle;
//------------------------------
      A     #Ma.CmdFaultReset;
      S     #DFxx.InCommand.CmdFaultResetAll;
//------------------------------
      A     #Ma.CmdSendB101;
      R     #Ma.CmdSendB101;
      S     #DFxx.In.CmdSendB101;
//------------------------------
      A     #Ma.CmdSendB102;
      R     #Ma.CmdSendB102;
      S     #DFxx.In.CmdSendB102;
//------------------------------
      A     #Ma.CmdSendB103;
      R     #Ma.CmdSendB103;
      S     #DFxx.In.CmdSendB103;
//------------------------------
      A     #Ma.CmdSendB104;
      R     #Ma.CmdSendB104;
      S     #DFxx.In.CmdSendB104;
NETWORK
TITLE = Digital outputs to DFCA
      A     #Ma.InpLL;
      =     #Ma.OutpLL;
      A     #Ma.InpLevelMiddle;
      =     #Ma.OutpLevelMiddle;
NETWORK
TITLE = Input signal from DP modul
      AN    #Ma.Par.ParDP;
      JC    IPJ0;
//===================================
      L     #DFxx.OutA101Ac.Mode;
      L     1;
      ==I;
      =     #ElRemote.InpTrue;
//===================================
      L     #DFxx.OutA101Ac.State;
      L     4;
      ==I;
      =     #ElRunning.InpTrue;
//===================================
      AN    #DFxx.OutA104Ac.SumAlarm;
      =     #ElSumFault.InpTrue;
IPJ0: NOP   0;
NETWORK
TITLE = Call Digital Input: ElRemote
      CALL  #ElRemote;
NETWORK
TITLE = Call Digital Input: ElRunning
      CALL  #ElRunning;
NETWORK
TITLE = Call Digital Input: ElSumFault
      CALL  #ElSumFault;
NETWORK
TITLE = Call Digital Input: ElFireAlarm
      CALL  #ElFireAlarm;
NETWORK
TITLE = Call ElPressStart
      CALL  #ElPressStart;
NETWORK
TITLE = Call ElDischargerRunning
      CALL  #ElDischargerRunning;
NETWORK
TITLE = Call Digital Input: ElDPFault
      ON    #Ma.Par.ParDP;
      ON    #DFxx.Out.DPFault;
      =     #ElDPFault.InpTrue;
      CALL  #ElDPFault;
NETWORK
TITLE = State
//-Relais contro:
// State:
// -Idle
// -Startup
// -Operation
// -Shutdown
//
      A     #ElRemote.StFault;
      O     #ElRunning.StFault;
      O     #ElSumFault.StFault;
      O     #ElFireAlarm.StFault;
      O     #ElPressStart.StFault;
      O     #ElDischargerRunning.StFault;
      O     #ElDPFault.StFault;
      =     #tmpFaultSum;
//=================================
//State StFault
//=================================
      A     #tmpFaultSum;
      =     #Ma.StFault;
//=================================
//State StIdle
//=================================
      L     #DFxx.OutA101Ac.State;
      L     0;
      ==I;
      A     #Ma.Par.ParDP;
      AN    #tmpFaultSum;
      O(;
      ON    #Ma.InpLL;
      ON    #Ma.InDischargerRunning;
      ON    #ElPressStart.StStarted;
      ON    #ElRemote.InpTrue;
      AN    #ElRunning.InpTrue;
      AN    #Ma.Par.ParDP;
      );
      =     #Ma.StIdle;
//=================================
//State StStartup
//=================================
      L     #DFxx.OutA101Ac.State;
      L     1;
      ==I;
      A     #Ma.Par.ParDP;
      AN    #tmpFaultSum;
      O(;
      AN    #Ma.StIdle;
      AN    #ElRunning.InpTrue;
      AN    #Ma.StFault;
      AN    #Ma.Par.ParDP;
      );
      =     #Ma.StStartup;
//=================================
//State StReady
//=================================
      L     #DFxx.OutA101Ac.State;
      L     2;
      ==I;
      A     #Ma.Par.ParDP;
      AN    #tmpFaultSum;
      =     #Ma.StReady;
//=================================
//State StFeedStartup
//=================================
      L     #DFxx.OutA101Ac.State;
      L     3;
      ==I;
      A     #Ma.Par.ParDP;
      AN    #tmpFaultSum;
      =     #Ma.StFeedStartup;
//=================================
//State StOperation
//=================================
      L     #DFxx.OutA101Ac.State;
      L     4;
      ==I;
      A     #Ma.Par.ParDP;
      AN    #tmpFaultSum;
      O(;
      AN    #Ma.Par.ParDP;
      A     #ElRunning.InpTrue;
      AN    #Ma.StIdle;
      AN    #Ma.StStartup;
      AN    #Ma.StFault;
      );
      =     #Ma.StOperation;
//=================================
//State StShutdown
//=================================
      L     #DFxx.OutA101Ac.State;
      L     5;
      ==I;
      A     #Ma.Par.ParDP;
      AN    #tmpFaultSum;
      O(;
      AN    #Ma.Par.ParDP;
      AN    #Ma.StIdle;
      AN    #Ma.StStartup;
      AN    #Ma.StFault;
      AN    #Ma.StOperation;
      );
      =     #Ma.StShutdown;
NETWORK
TITLE = Global End
      CLR;	//---Clear all commands
      =     #Ma.CmdOn;
      =     #Ma.CmdOff;
      =     #Ma.CmdNext;
      =     #Ma.CmdFaultReset;
      =     #Ma.CmdResetHorn;
NETWORK
TITLE = Digital outputs Lamp
//-----------------------------
      A     #ElRunning.InpTrue;
      =     #Ma.OutpLampRunning;
//-----------------------------
      AN    #ElSumFault.InpTrue;
      =     #Ma.OutpLampFault;
//-----------------------------
      AN    #ElFireAlarm.InpTrue;
      =     #Ma.OutpLampFireAlarm;
NETWORK
TITLE = State Code
// Same as motor
      A     #Ma.StIdle;
      L     1;	//  StCode 1=StIdle
      JC    Code;
      A     #Ma.StStartup;
      L     2;	//  StCode 2=StStartup
      JC    Code;
      A     #Ma.StReady;
      L     3;	//  StCode 3=StReady
      JC    Code;
      A     #Ma.StFeedStartup;
      L     4;	//  StCode 4=StFeedStartup
      JC    Code;
      A     #Ma.StOperation;
      L     5;	//  StCode 5=StOperation
      JC    Code;
      A     #Ma.StShutdown;
      L     6;	//  StCode 6=StShutdown
      JC    Code;
      L     32;	// StCode=Fault
Code: L     #Ma.StCode;	// Old state code
      TAK;
      T     #Ma.StCode;	// Save state code
      <>I;
      L     3;
      CC    "SYS_CBitCtrl";	//Set change bit
END_FUNCTION_BLOCK

FUNCTION_BLOCK "GCS7_M_MYFB"	// FB 64
TITLE = Machine MYEB Moisture Control
//  
//COPYRIGHT:    (C) 1997  BUHLER AG, CH-9240 UZWIL, SWITZERLAND
//
//PRODUCT:      GCS7
//
//TITLE:        Machine MYEB Moisture Control
//
//-------------------------------------------------------------------------
//
//IDENT:        AUTHOR:             DEPT:                      DATE:
//
//FB64.4.2      A. Egli             CT3                        02-Jul-2004
//              Run delay time water also when MOZ_DosingEnable is StStopped
//FB64.4.1      A. Egli             CT3                        24-Jun-2004
//              InDisableConveyor
//              FB64.3.3 GCS90S7 : InLocalWaterControl 
//FB64.4.0      A. Egli             CT3                        17-Jun-2002
//              New Release with one block 
//FB64.3.2      Ph. Engler          MU664                      19-Feb-2002
//              _Product flowmonitor: CmdRunTimeoutTime integrated
//FB64.3.1      A.Egli              CT3                        30-Oct-2001
//              InDisableWater
//FB64.3.0      S. Kalberer         CT3                        11-Oct-1999
//              Local data reduced
//FB64.2B       S. Kalberer         CT3                        10-Aug-1998
//              Clear CmdNewValue/CmdNewJob adjusted
//FB64.2A       A. Egli             CT3                        04-Mai-1998
//              StFault = StCode 32
//FB64.1A       S. Kalberer         AEE61                      22-Oct-1997
//              1st Release in S7
//
//-------------------------------------------------------------------------
//
//PURPOSE:      MANUAL : see [LL.MYBxxMAN]
//
//RESTRICTIONS: S7
//              ACCU2: Pointer to dynamic datas of the element
//              ACCU1: Pointer to parameter datas of the element
//
//-------------------------------------------------------------------------
//
AUTHOR : EA
FAMILY : GCS7LL
NAME : MYEB_Ma
VERSION : 4.2
VAR
  Ma : UDT 20640;
  MYEB_LC : FB 23;	//Element
  MYEB_GroupAlarm : FB 14;	//Element
  MYF_Product : FB 14;	//Element
  MYF_ConveyorEnable : FB 11;	//Element
  MOZ_DosingEnable : FB 11;	//Element
  MOZ_WaterValve : FB 11;	//Element
  MOZ_Product : FB 14;	//Element
  MOZ_Motor : FB 12;	//Element
END_VAR
VAR_TEMP
  tmpLenDyn : DINT ;
  tmpFaultSum : BOOL ;
  tmpFaultReset : BOOL ;
END_VAR
BEGIN
NETWORK
TITLE =
      L     30;
      T     #tmpLenDyn;	//--> Len dynamic data in byte
NETWORK
TITLE = PC Control
//=== Test Object number =====================
      L     "SYS_DirectCtrlDB".PC.ObjectNo;	//PCControl.ObjectNo
      L     #Ma.Par.ParObjectNo;	//Input ObjectNo
      <>I;
      JC    aEnd;
//=== Test OType      ========================
      L     2064;	//Input object type
      L     "SYS_DirectCtrlDB".PC.ObjectType;	//PCControl.ObjectType
      <>I;
      JC    aEnd;
//=== Test Handshake =========================
      A     "SYS_DirectCtrlDB".PC.Hsk.FExamine;	// Handshake.FExamine
      JC    aExa;
      A     "SYS_DirectCtrlDB".PC.Hsk.FDefineCmd;	// Handshake.FDefineCmd
      JC    aCmd;
      A     "SYS_DirectCtrlDB".PC.Hsk.FDefinePara;	// Handshake.FDefinePara
      JC    pPar;
aIni: L     2;	// FcInit
      UC    "SYS_DirectCtrl";
      JU    aEnd;
// Write parameter 
pPar: LAR1  P#DBX 58.0;
      L     P#6.0;
      +AR1;
      L     DBW [AR1,P#4.0];
      T     #Ma.Par.ParStartValuePc;
      L     DBW [AR1,P#6.0];
      T     #Ma.Par.ParStartValue;
      L     DBW [AR1,P#8.0];
      T     #Ma.Par.ParOffDelayFeed;
      L     DBW [AR1,P#10.0];
      T     #Ma.Par.ParOnDelayWater;
// Write new commands from PC to Interface of group 
aCmd: A     "SYS_DirectCtrlDB".PC.Cmd1[4];	//Cmd1[4]=CmdNewValue
      S     #Ma.CmdNewValue;
      A     "SYS_DirectCtrlDB".PC.Cmd1[5];	//Cmd1[5]=CmdNewJob
      S     #Ma.CmdNewJob;
      A     "SYS_DirectCtrlDB".PC.Cmd1[8];	//Cmd1[8]=CmdOff
      S     #Ma.CmdOff;
      A     "SYS_DirectCtrlDB".PC.Cmd1[9];	//Cmd1[9]=CmdOn
      S     #Ma.CmdOn;
      A     "SYS_DirectCtrlDB".PC.Cmd1[10];	//Cmd1[10]=CmdNext
      S     #Ma.CmdNext;
      A     "SYS_DirectCtrlDB".PC.Cmd1[11];	//Cmd1[11]=CmdFaultReset
      S     #Ma.CmdFaultReset;
      A     "SYS_DirectCtrlDB".PC.Cmd1[13];	//Cmd1[13]=CmdManualOn
      S     #Ma.InManual;
      A     "SYS_DirectCtrlDB".PC.Cmd1[15];	//Cmd1[15]=CmdManualWaterOn
      S     #Ma.InManualWaterControl;
      A     "SYS_DirectCtrlDB".PC.Cmd2[13];	//Cmd2[13]=CmdManualOff
      R     #Ma.InManual;
      A     "SYS_DirectCtrlDB".PC.Cmd2[15];	//Cmd2[15]=CmdManualWaterOff
      R     #Ma.InManualWaterControl;
      JU    aIni;
aExa: TAR2;	// Address Dynamic datas
      T     "SYS_DirectCtrlDB".GC.InDynAddr;	// -->PCControl.GC.InDynAddr
      L     #tmpLenDyn;	// Length Dynamic datas
      T     "SYS_DirectCtrlDB".GC.InDynLen;	// -->PCControl.GC.InDynLen
      L     0;
      T     "SYS_DirectCtrlDB".GC.InParaAddr;	// -->PCControl.GC.InParaAddr
      T     "SYS_DirectCtrlDB".GC.InParaLen;	// -->PCControl.GC.InParaLen
      L     1;	// Code FcExamine
      UC    "SYS_DirectCtrl";
      L     10;	//Revision
      T     "SYS_DirectCtrlDB".GC.Revision;
aEnd: NOP   0;
NETWORK
TITLE =  Timer switch off feed and switch on water
//Timer switch off delay feed
      A     #MOZ_WaterValve.StStarted;
      AN    #Ma.OutMoistureStart;
      A     #Ma.OutFeedReady;
      AN    #Ma.InProductFeed;
      JC    TiF0;
      R     #Ma.OutOffDelayFeedRun;
      L     0;	//Reset timervalue to zero
      T     #Ma.Par.OutOffDelayFeed;
      JU    TiW;
TiF0: A     #Ma.OutOffDelayFeedDone;
      JC    TiW;
      A     #Ma.OutOffDelayFeedRun;
      JC    TiF1;
      S     #Ma.OutOffDelayFeedRun;
      L     #Ma.Par.ParOffDelayFeed;
      T     #Ma.Par.OutOffDelayFeed;
TiF1: AN    "GCS7_Gr_OutTick1s";	//Gr.OutTick1S
      L     #Ma.Par.OutOffDelayFeed;
      JC    TiF2;
      +     -10;
      T     #Ma.Par.OutOffDelayFeed;
TiF2: L     0;
      <=I;
      R     #Ma.OutOffDelayFeedRun;
      S     #Ma.OutOffDelayFeedDone;
TiW:  A     #MOZ_Product.StTrue;
      O     #MOZ_Product.StCtoTrue;
      A(;	//[4.2]
      A     #MOZ_WaterValve.StStopped;
      O     #MOZ_DosingEnable.StStopped;	//[4.2]
      );	//[4.2]
      A     #Ma.OutFeedReady;
      A     #Ma.InProductFeed;
      JC    TiW0;
      R     #Ma.OutOnDelayWaterRun;
      L     0;	//Reset timervalue to zero
      T     #Ma.Par.OutOnDelayWater;
      JU    TiE;
//Timer swtich on delay water
TiW0: A     #Ma.OutOnDelayWaterDone;
      JC    TiE;
      A     #Ma.OutOnDelayWaterRun;
      JC    TiW1;
      S     #Ma.OutOnDelayWaterRun;
      L     #Ma.Par.ParOnDelayWater;
      T     #Ma.Par.OutOnDelayWater;
TiW1: AN    "GCS7_Gr_OutTick1s";	//Gr.OutTick1S
      L     #Ma.Par.OutOnDelayWater;
      JC    TiW2;
      +     -10;
      T     #Ma.Par.OutOnDelayWater;
TiW2: L     0;
      <=I;
      R     #Ma.OutOnDelayWaterRun;
      S     #Ma.OutOnDelayWaterDone;
//---Reset timer Done bit
TiE:  AN    #Ma.InProductFeed;
      O     #MOZ_Product.StFalse;
      R     #Ma.OutOnDelayWaterDone;
      A     #Ma.InProductFeed;
      R     #Ma.OutOffDelayFeedDone;
NETWORK
TITLE =  Set moisture StartValue or StartValuePc [%]
      A     #Ma.InManualWaterControl;
      O     #Ma.InLocalWaterControl;	//[3.3] InLocalWaterControl
      O     #Ma.StStopped;
      ON    #Ma.InProductFeed;
      ON    #Ma.Par.ParWithMYEB_LC;
      R     #Ma.OutMoistureStart;
      JC    MoSE;
      AN    #MOZ_Product.StTrue;	//Condition for new dosing offset
      AN    #MOZ_Product.StCtoFalse;
      O     #MYF_Product.StTrue;
      O     #MYF_Product.StCtoFalse;
      O     #Ma.OutMoistureStartPc;
      JC    MoS1;
      S     #Ma.OutMoistureStart;
      S     #Ma.OutMoistureStartPc;
      S     #Ma.CmdNewValue;
      S     #MYEB_LC.CmdNewValue;	//[4.1]B
      L     #Ma.Par.ParStartValuePc;
      ITD;	// 16bit --> 32bit
      DTR;	// 32bit-DINT --> REAL
      L     1.000000e+02;
      /R;
      L     #Ma.Par.ParStartValue;
      DTR;
      *R;
      RND;	// REAL --> 32bit-DINT
      T     #MYEB_LC.InStartValue;
      JU    MoSE;
MoS1: AN    #MYF_Product.StTrue;
      AN    #MYF_Product.StCtoFalse;
      ON    #Ma.OutMoistureStartPc;
      JC    MoSE;
      R     #Ma.OutMoistureStartPc;
      S     #Ma.CmdNewValue;
      S     #MYEB_LC.CmdNewValue;	//[4.1]B
      L     #Ma.Par.ParStartValue;
      T     #MYEB_LC.InStartValue;
MoSE: NOP   0;
NETWORK
TITLE = Interlocking
//===Clear tmp Variable
//
//===Global Group Orders===
//---FaultReset is on---
      A     "GCS7_Gr_OutFaultReset";	//Gr.OutFaultReset
      O     #Ma.CmdFaultReset;
      =     #tmpFaultReset;
//---Manual Mode---
      A     "GCS7_Gr_OutManualOn";	//Gr.OutManualOn
      S     #Ma.InManual;
      A     "GCS7_Gr_OutManualOff";	//Gr.OutManualOff
      R     #Ma.InManual;
      A     #Ma.InManual;
      S     "GCS7_Gr_InManual";	//Gr.InManual
//--- Fault----
      A     #MYEB_LC.StFault;
      A     #Ma.Par.ParWithMYEB_LC;
      O;
      A     #MYEB_GroupAlarm.StFault;
      A     #Ma.Par.ParWithMYEB_GroupAlarm;
      O     #MYF_Product.StFault;
      O;
      A     #MYF_ConveyorEnable.StFault;
      A     #Ma.Par.ParWithMYF_Conveyor;
      O     #MOZ_DosingEnable.StFault;
      O     #MOZ_WaterValve.StFault;
      O     #MOZ_Product.StFault;
      O     #MOZ_Motor.StFault;
      =     #tmpFaultSum;
//--- Fault Reset -------------
      A     #tmpFaultReset;
      A     #tmpFaultSum;
      S     #MYEB_LC.CmdFaultReset;
      S     #MYEB_GroupAlarm.CmdFaultReset;
      S     #MYF_Product.CmdFaultReset;
      S     #MYF_ConveyorEnable.CmdFaultReset;
      S     #MOZ_DosingEnable.CmdFaultReset;
      S     #MOZ_WaterValve.CmdFaultReset;
      S     #MOZ_Product.CmdFaultReset;
      S     #MOZ_Motor.CmdFaultReset;
//===Element interlocking===
//--- MYF_CoveyorEnable ----
      A     #Ma.Par.ParWithMYF_Conveyor;
      A     #Ma.InEnable;
      AN    #Ma.InLocal;
      AN    #Ma.InDisableConveyor;	//[4.1]
      =     #MYF_ConveyorEnable.InEnable;
//--- MOZ_Motor ----
      A     #Ma.InEnable;
      =     #MOZ_Motor.InEnableFwd;
//+++Feeding ready+++
      A     #MYF_ConveyorEnable.StStarted;
      ON    #Ma.Par.ParWithMYF_Conveyor;
      O     #Ma.InManualWaterControl;
      A     #MOZ_Motor.StStartedFwd;
      =     #Ma.OutFeedReady;
//---MOZ_DosingEnable---
      A     #MOZ_Product.StTrue;
      O     #MOZ_Product.StCtoFalse;
      A     #Ma.OutFeedReady;
      A(;
      O     #Ma.OutOnDelayWaterDone;
      O     #Ma.OutOffDelayFeedRun;
      );
      A(;
      ON    #Ma.OutMoistureStart;
      ON    #MYEB_LC.OutNewValueActive;
      );
      AN    #tmpFaultSum;
      AN    #Ma.InManualWaterControl;
      AN    #Ma.InDisableWaterDosing;	//[3.1]
      AN    #Ma.InDisableConveyor;	//[4.1]
      A     #Ma.InEnable;
      AN    #Ma.InLocal;
      =     #MOZ_DosingEnable.InEnable;
      A     #MOZ_DosingEnable.StStopped;	//[4.2]
      S     #MOZ_DosingEnable.CmdNext;
//---MOZ_WaterValve---
      A     #MOZ_Product.StTrue;
      O     #MOZ_Product.StCtoFalse;
      A     #Ma.OutFeedReady;
      A(;
      O     #Ma.OutMoistureStart;
      O     #MOZ_DosingEnable.InEnable;
      O     #Ma.OutOnDelayWaterDone;
      O     #Ma.OutOffDelayFeedRun;
      );
      AN    #Ma.InDisableWaterDosing;	//[3.1]
      AN    #Ma.InDisableConveyor;	//[4.1]
      AN    #tmpFaultSum;
      AN    #Ma.InLocal;
      =     #MOZ_WaterValve.InEnable;
      S     #MOZ_WaterValve.CmdNext;
//---Set CmdNext---
      A     #Ma.CmdOn;
      A     #Ma.InManual;
      O;
      A     #Ma.CmdNext;
      AN    #Ma.InManual;
      S     #MYF_ConveyorEnable.CmdNext;
      S     #MOZ_Motor.CmdNext;
//---Set CmdOff---
      A     #Ma.CmdOff;
      S     #MYF_ConveyorEnable.CmdOff;
      S     #MOZ_Motor.CmdOff;
      S     #MOZ_WaterValve.CmdOff;
      S     #MOZ_DosingEnable.CmdOff;
//--- Local&ManualWater mode --
      A     #Ma.InLocal;	//[3.3]
      O     #Ma.InManualWaterControl;	//[3.3]
      O     #Ma.InLocalWaterControl;	//[3.3] InLocalWaterControl
      =     #MYEB_LC.InLocal;	//[3.3]
      =     #MYEB_GroupAlarm.InLocal;	//[3.3]
      A     #Ma.InLocal;
      O     #Ma.InManualWaterControl;
//[3.3]      =     #MYEB_LC.InLocal     
//[3.3]      =     #MYEB_GroupAlarm.InLocal
      =     #MYF_ConveyorEnable.InLocal;
      =     #MOZ_DosingEnable.InLocal;
      A     #Ma.InLocal;
      =     #MOZ_Motor.InLocal;
      =     #MOZ_WaterValve.InLocal;
      =     #MOZ_Product.InLocal;
      =     #MYF_Product.InLocal;
//---Switch on monitoring the digital input
      A     #Ma.Par.ParWithMYEB_GroupAlarm;
      =     #MYEB_GroupAlarm.InMonTrue;
      A     #Ma.InEnable;
      A     #Ma.InProductFeed;
      FP    #MOZ_Product.InMonTrue;	// [3.2]  ( =  -> FP)
      S     #MOZ_Product.CmdRunTimeoutTime;	// [3.2]
      A     #Ma.InEnable;
      A     #Ma.InProductFeed;
      AN    #Ma.InManualWaterControl;
      FP    #MYF_Product.InMonTrue;	// [3.2]  ( =  -> FP)
      S     #MYF_Product.CmdRunTimeoutTime;	// [3.2]
NETWORK
TITLE =  Call MYEB Moisture Control Unit: MYEB_LC
      AN    #Ma.Par.ParWithMYEB_LC;
      JC    MYEB;
//---Interlocking
      AN    #Ma.OutMoistureStart;	//[4.1]B
      AN    #MYEB_LC.OutNewValueActive;	//[4.1]B
      A     #Ma.CmdNewValue;
      AN    #MYEB_LC.CmdNewValue;	//2B:
      R     #Ma.CmdNewValue;
      S     #MYEB_LC.CmdNewValue;
      AN    #MYEB_LC.CmdNewValue;
      AN    #MYEB_LC.OutNewValueActive;
      AN    #Ma.OutMoistureStartPc;
      A     #Ma.OutMoistureStart;	//[4.1]B
      R     #Ma.OutMoistureStart;
      A     #Ma.CmdNewJob;
      AN    #MYEB_LC.CmdNewJob;	//2B:
      R     #Ma.CmdNewJob;
      S     #MYEB_LC.CmdNewJob;
//---calling the element
      CALL  #MYEB_LC;
NETWORK
TITLE = Call Digital Input: MYEB_GroupAlarm 
MYEB: AN    #Ma.Par.ParWithMYEB_GroupAlarm;
      JC    MYFB;
      CALL  #MYEB_GroupAlarm;
NETWORK
TITLE = Call Digital Input: MYF_Product
MYFB: CALL  #MYF_Product;
NETWORK
TITLE = Call Digital Output: MYFConveyorEnable
      AN    #Ma.Par.ParWithMYF_Conveyor;
      JC    MOZ;
      CALL  #MYF_ConveyorEnable;
NETWORK
TITLE = Call Digital Output: MOZDosingEnable
MOZ:  CALL  #MOZ_DosingEnable;
NETWORK
TITLE = Call Digital Output: MOZWaterValve
      CALL  #MOZ_WaterValve;
NETWORK
TITLE = Call Digital Input: MOZ_Product
      CALL  #MOZ_Product;
NETWORK
TITLE = Call Motor Control: MOZ_Motor
      CALL  #MOZ_Motor;
NETWORK
TITLE = Jump to actual state
//===State machine===
      A     #Ma.StStopped;
      JC    S0;
      A     #Ma.StStarted;
      JC    S2;
      A     #Ma.StStarting;
      JC    S1;
      A     #Ma.StStopping;
      JC    S3;
      A     #Ma.StFault;
      JC    S4;
NETWORK
TITLE = Stopped
//any Transition 
xxS0: S     #Ma.StStopped;
      JU    OUT;
//=== Logic
// Condition for StFault
S0:   A     #tmpFaultSum;
      R     #Ma.StStopped;
      JC    xxS4;	//--> ST_FAULT:
// Condition for StStarting
      AN    #MYF_ConveyorEnable.StStopped;
      AN    #MYF_ConveyorEnable.StFalse;
      A     #Ma.Par.ParWithMYF_Conveyor;
      ON    #MOZ_Motor.StStopped;
      R     #Ma.StStopped;
      JC    xxS1;	//--> StStarting
      JU    OUT;
NETWORK
TITLE = StStarting
//any Transition 
xxS1: S     #Ma.StStarting;
      JU    OUT;
//=== Logic
// Condition for StFault
S1:   A     #tmpFaultSum;
      R     #Ma.StStarting;
      JC    xxS4;	//--> StFault
// Condition for StStopping
      A     #MYF_ConveyorEnable.StStopped;
      ON    #Ma.Par.ParWithMYF_Conveyor;
      A     #MOZ_Motor.StStopped;
      R     #Ma.StStarting;
      JC    xxS3;	//-->StStopping
// Condition for StStarted
      A     #Ma.OutFeedReady;
      R     #Ma.StStarting;
      JC    xxS2;	//-->StStarted
      JU    OUT;
NETWORK
TITLE = StStarted
//any Transition 
xxS2: S     #Ma.StStarted;
      JU    OUT;
//=== Logic
// Condition for StFault
S2:   A     #tmpFaultSum;
      R     #Ma.StStarted;
      JC    xxS4;	//--> StFault
// Condition for StStopping
      A     #MYF_ConveyorEnable.StStopped;
      A     #Ma.Par.ParWithMYF_Conveyor;
      AN    #Ma.InManualWaterControl;
      AN    #Ma.InDisableConveyor;	//[4.1]
      ON    #MOZ_Motor.StStartedFwd;
      R     #Ma.StStarted;
      JC    xxS3;	//-->StStopping
      JU    OUT;
NETWORK
TITLE = Stopping
//any Transition 
xxS3: S     #Ma.StStopping;
      JU    OUT;
//=== Logic
// Condition for StFault
S3:   A     #tmpFaultSum;
      R     #Ma.StStopping;
      JC    xxS4;	//--> StFault
// Condition for StStopped
      A     #MYF_ConveyorEnable.StStopped;
      O     #MYF_ConveyorEnable.StFalse;
      ON    #Ma.Par.ParWithMYF_Conveyor;	//Element used?
      A     #MOZ_DosingEnable.StStopped;
      A     #MOZ_WaterValve.StStopped;
      A     #MOZ_Motor.StStopped;
      R     #Ma.StStopping;
      JC    xxS0;	//-->StStopped
// Condition for StStarting
      AN    #MYF_ConveyorEnable.StStopped;
      AN    #MYF_ConveyorEnable.StFalse;
      ON    #Ma.Par.ParWithMYF_Conveyor;	//Element used?
      O     #Ma.InDisableConveyor;	//[4.1]
      O     #Ma.InManualWaterControl;	//[3.3][4.1]
      AN    #MOZ_Motor.StStopped;
      AN    #MOZ_Motor.StStopping;
      R     #Ma.StStopping;
      JC    xxS1;	//-->StStarting
      JU    OUT;
NETWORK
TITLE = Fault
//any Transition 
xxS4: S     #Ma.StFault;
      JU    OUT;
//=== Logic
S4:   A     #tmpFaultSum;
      AN    #tmpFaultReset;
      AN    #Ma.InLocal;
      JC    OUT;
// Condition for StStopping
      AN    #tmpFaultSum;
      R     #Ma.StFault;
      JC    xxS3;	//-->StStopping
      JU    OUT;
NETWORK
TITLE = Global End
OUT:  CLR;	//---Clear all commands
      =     #Ma.CmdOn;
      =     #Ma.CmdOff;
      =     #Ma.CmdNext;
      =     #Ma.CmdFaultReset;
NETWORK
TITLE = State Code
// State                 StCode    
// -----------------------------
// StFault                  32
// StStopped                1
// StStarting               2
// StStartedWait            3
// StStopping               4
// StStartedMoistureStart   5
// StStartedMoisture        6
      A     #Ma.StStopped;
      L     1;	// Code: stopped
      JC    STC9;
      A     #Ma.StStarting;
      L     2;	// Code: starting
      JC    STC9;
      A     #Ma.OutMoistureStart;
      A     #Ma.OutFeedReady;
      L     5;	// Code: started moisture start
      JC    STC9;
      A     #MOZ_DosingEnable.StStarted;
      O     #Ma.InManualWaterControl;
      A     #MOZ_WaterValve.StStarted;
      A     #Ma.OutFeedReady;
      L     6;	// Code: started moisture
      JC    STC9;
//[4.1]      U     #Ma.OutFeedReady
      A     #Ma.StStarted;	//[4.1]
      L     3;	// Code: started wait
      JC    STC9;
      A     #Ma.StStopping;
      L     4;	// Code: stopping
      JC    STC9;
      L     32;	// 2A: Code: fault
STC9: L     #Ma.StCode;	// Old state code
      TAK;
      T     #Ma.StCode;	// Save state code
      <>I;
      L     3;	// Load code for CBit methode
      CC    "SYS_CBitCtrl";
END_FUNCTION_BLOCK

FUNCTION_BLOCK "GCS7_M_PulsePhaseConv"	// FB 65
TITLE = Pulse Phase Conveying system
//  
//COPYRIGHT:    (C) 1997  BUHLER AG, CH-9240 UZWIL, SWITZERLAND
//
//PRODUCT:      GCS7
//
//TITLE:        FB 65 Machine Control:Pulse Phase Conveying System
//
//Revision:     GCPROVB Revision 11
//
//-------------------------------------------------------------------------
//
//IDENT:        AUTHOR:             DEPT:                       DATE:
//
//FB65.5.0      A. Egli             CT3                         11-Apr-2008
//              Air Vessel
//FB65.4.1      A. Egli             CT3                         16-Feb-2006
//              HL.InpMonFalse only when level is covered
//FB65.4.0      A. Egli             CT3                         17-Jun-2002
//              New Release with one block 
//FB65.3.0      A. Egli             CT3                         11-Oct-1999
//              Local data reduced
//FB65.2C       A. Egli             CT3                         26-Mai-1999
//              Reset OutClearingPulsingEnd by transition to StStarting 
//FB65.2B       K. Tischer          MU664                       06-Mrz-1999
//              CC FC2 not UC FC2
//FB65.2A       A. Egli             CT3                         04-Mai-1998
//              StFault = StCode 32
//FB65.1A       A.Egli              AEE61                       15-Oct-1997
//              1st Release in S7
//
//-------------------------------------------------------------------------
//
//PURPOSE:      MANUAL : see [LL.TAKxxMAN]
//
//RESTRICTIONS: S7
//              ACCU2: Pointer to dynamic datas of the machine
//              ACCU1: Pointer to parameter datas of the machine
//
//-------------------------------------------------------------------------
//
AUTHOR : EA
FAMILY : GCS7LL
NAME : PulsePha
VERSION : 5.0
VAR
  Ma : UDT 20650;
  Airlock : FB 12;	//Element
  Pressure : FB 16;	//Element
  MainValve : FB 13;	//Element
  MatValve : FB 13;	//Element
  AirValve : FB 13;	//Element
  BypassValve : FB 13;	//Element
  SpeedMon : FB 14;	//Element
  HL : FB 14;	//Element
  ClearingValve : FB 13;	//Element
END_VAR
VAR_TEMP
  tmpEnable : BOOL ;
  tmpFaultStop : BOOL ;
  tmpFaultValve : BOOL ;
  tmpFaultTime : BOOL ;
  tmpStoppedMan : BOOL ;
  tmpReadyConveying : BOOL ;
  tmpClosingDelayEnd : BOOL ;
  tmpClearing : BOOL ;
  tmpVKE : BOOL ;
  tmpLenDyn : INT ;
  tmpCleared : BOOL ;
END_VAR
BEGIN
NETWORK
TITLE =
      L     60;
      T     #tmpLenDyn;
NETWORK
TITLE = PC Control
//=== Test Object number =====================
      L     "SYS_DirectCtrlDB".PC.ObjectNo;	//PCControl.ObjectNo
      L     #Ma.Par.ParObjectNo;	//Input ObjectNo
      <>I;
      JC    aEnd;
//=== Test OType      ========================
      L     2065;	//Input object type
      L     "SYS_DirectCtrlDB".PC.ObjectType;	//PCControl.ObjectType
      <>I;
      JC    aEnd;
//=== Test Handshake =========================
      A     "SYS_DirectCtrlDB".PC.Hsk.FExamine;	// Handshake.FExamine
      JC    aExa;
      A     "SYS_DirectCtrlDB".PC.Hsk.FDefineCmd;	// Handshake.FDefineCmd
      JC    aCmd;
      A     "SYS_DirectCtrlDB".PC.Hsk.FDefinePara;	// Handshake.FDefinePara
      JC    pPar;
aIni: L     2;	// FcInit
      UC    "SYS_DirectCtrl";
      JU    aEnd;
// Write parameter 
pPar: LAR1  P#DBX 58.0;
      L     P#6.0;
      +AR1;
      L     DBW [AR1,P#4.0];
      T     #Ma.Par.ParDelayMain;
      L     DBW [AR1,P#6.0];
      T     #Ma.Par.ParDelayAirlock;
      L     DBW [AR1,P#8.0];
      T     #Ma.Par.ParPulseMatTime;
      L     DBW [AR1,P#10.0];
      T     #Ma.Par.ParPulseAirTime;
      L     DBW [AR1,P#12.0];
      T     #Ma.Par.ParClearingPulsing;
      L     DBW [AR1,P#14.0];
      T     #Ma.Par.ParClearingBoth;
      L     DBW [AR1,P#16.0];
      T     #Ma.Par.ParClearingBypass;
      L     DBW [AR1,P#18.0];
      T     #Ma.Par.ParDelayClosing;
// Write new commands from PC to Interface of group 
aCmd: A     "SYS_DirectCtrlDB".PC.Cmd1[8];	//Cmd1[8]=CmdOff
      S     #Ma.CmdOff;
      A     "SYS_DirectCtrlDB".PC.Cmd1[9];	//Cmd1[9]=CmdMainOnOff
      S     #Ma.CmdMainOnOff;
      A     "SYS_DirectCtrlDB".PC.Cmd1[3];	//Cmd1[3]=CmdAirlockOnOff
      S     #Ma.CmdAirlockOnOff;
      A     "SYS_DirectCtrlDB".PC.Cmd1[4];	//Cmd1[3]=CmdOpenAll
      S     #Ma.CmdOpenAll;
      A     "SYS_DirectCtrlDB".PC.Cmd1[5];	//Cmd1[3]=CmdPulsingOnOff
      S     #Ma.CmdPulsingOnOff;
      A     "SYS_DirectCtrlDB".PC.Cmd1[10];	//Cmd1[10]=CmdNext
      S     #Ma.CmdNext;
      A     "SYS_DirectCtrlDB".PC.Cmd1[11];	//Cmd1[11]=CmdFaultReset
      S     #Ma.CmdFaultReset;
      A     "SYS_DirectCtrlDB".PC.Cmd1[13];	//Cmd1[13]=CmdManualOn
      S     #Ma.InManual;
      A     "SYS_DirectCtrlDB".PC.Cmd2[13];	//Cmd2[13]=CmdManualOff
      R     #Ma.InManual;
      JU    aIni;
aExa: TAR2;	// Address Dynamic datas
      T     "SYS_DirectCtrlDB".GC.InDynAddr;	// -->PCControl.GC.InDynAddr
      L     #tmpLenDyn;	// Length Dynamic datas
      T     "SYS_DirectCtrlDB".GC.InDynLen;	// -->PCControl.GC.InDynLen
      L     0;
      T     "SYS_DirectCtrlDB".GC.InParaAddr;	// -->PCControl.GC.InParaAddr
      T     "SYS_DirectCtrlDB".GC.InParaLen;	// -->PCControl.GC.InParaLen
      L     1;	// Code FcExamine
      UC    "SYS_DirectCtrl";
      L     11;	//Revision
      T     "SYS_DirectCtrlDB".GC.Revision;
aEnd: NOP   0;
NETWORK
TITLE = Interlocking
//===Global Group Orders===
//===Global Group Orders===
      A     "GCS7_Gr_OutManualOn";	///Gr.OutManualOn
      S     #Ma.InManual;
      A     "GCS7_Gr_OutManualOff";	//Gr.OutManualOff
      R     #Ma.InManual;
      A     #Ma.InManual;
      S     "GCS7_Gr_InManual";	//Gr.InManual
//Local
      A     #Ma.InLocal;
      AN    #Ma.InManual;
      =     #Airlock.InLocal;
      =     #MainValve.InLocal;
      =     #MatValve.InLocal;
      =     #AirValve.InLocal;
      =     #BypassValve.InLocal;
      =     #HL.InLocal;
      =     #SpeedMon.InLocal;
      =     #Pressure.InLocal;
      =     #ClearingValve.InLocal;	//[5.0]
//Enable 
      AN    #Ma.InLocal;
      A     #Ma.InEnable;
      O     #Ma.InManual;
      AN    #Ma.CmdOff;
      =     #tmpEnable;
      A     #Ma.InClearing;
      AN    #Ma.InManual;
      =     #tmpClearing;
//Monitoring 
      A     #Airlock.StStartedFwd;
      =     #SpeedMon.InMonTrue;
      A     #HL.InpTrue;	//[4.1]
      =     #HL.InMonFalse;
//Fault 
      O     #MainValve.StFault;
      O     #MatValve.StFault;
      O     #AirValve.StFault;
      O     #BypassValve.StFault;
      O     #ClearingValve.StFault;	//[5.0]
      =     #tmpFaultValve;
      A     #tmpFaultValve;
      O     #Pressure.StFault;
      =     #tmpFaultStop;
      A     #tmpFaultStop;
      O     #HL.StFault;
      O     #Airlock.StFault;
      O     #SpeedMon.StFault;
      =     #Ma.OutFault;
// Test stopped
      A     #Airlock.StStopped;
      A(;
      A     #MainValve.StLN;
      ON    #Ma.Par.ParWithMainValve;
      );
      A(;
      A     #MatValve.StLN;
      ON    #Ma.Par.ParWithMatValve;
      );
      A(;
      A     #AirValve.StLN;
      ON    #Ma.Par.ParWithAirValve;
      );
      A(;
      A     #BypassValve.StLN;
      ON    #Ma.Par.ParWithBypassValve;
      );
      A(;	//[5.0]
      A     #ClearingValve.StLN;	//[5.0]
      ON    #Ma.Par.ParWithClearingValve;	//[5.0]
      );	//[5.0]
      =     #tmpStoppedMan;
NETWORK
TITLE = Call Airlock
      CALL  #Airlock;
NETWORK
TITLE = Call PRange: Pressure
      CALL  #Pressure;
NETWORK
TITLE = Call Main Valve
      AN    #Ma.Par.ParWithMainValve;
      JC    El2;
      CALL  #MainValve;
NETWORK
TITLE = Call MatValve
El2:  AN    #Ma.Par.ParWithMatValve;
      JC    El3;
      CALL  #MatValve;
NETWORK
TITLE = Call AirValve
El3:  AN    #Ma.Par.ParWithAirValve;
      JC    El4;
      CALL  #AirValve;
NETWORK
TITLE = Call BypassValve
El4:  AN    #Ma.Par.ParWithBypassValve;
      JC    El5;
      CALL  #BypassValve;
NETWORK
TITLE = Call SpeedMon
El5:  AN    #Ma.Par.ParWithSpeedMon;
      JC    El6;
      CALL  #SpeedMon;
NETWORK
TITLE = Call HL
El6:  AN    #Ma.Par.ParWithHL;
      JC    El7;
      CALL  #HL;
NETWORK
TITLE = Call AirVesselValve
El7:  NOP   0;
      AN    #Ma.Par.ParWithClearingValve;
      JC    El8;
      CALL  #ClearingValve;
El8:  NOP   0;
NETWORK
TITLE = Jump to actual state
      A     #Ma.StStopped;
      JC    S0;
      A     #Ma.StStarting;
      JC    S1;
      A     #Ma.StStarted;
      JC    S2;
      A     #Ma.StFeeding;
      JC    S6;
      A     #Ma.StClearing;
      JC    S5;
      A     #Ma.StStopping;
      JC    S3;
NETWORK
TITLE = Stopped
//any Transition 
xxS0: S     #Ma.StStopped;	// ===> Initialisation
      JU    OUT;
//=== Logic
//Condition for Starting
S0:   AN    #Ma.InManual;
      AN    #Ma.InLocal;	//[5.0]
      A     #Ma.InEnable;
      A(;
      AN    #Ma.InClearing;
      O     #Ma.OutLoaded;	//[5.0]
      );
      A     #Ma.CmdNext;
      AN    #tmpFaultStop;
      ON    #tmpStoppedMan;
      R     #Ma.StStopped;
      JC    xxS1;	//-->StStarting
      JU    OUT;
NETWORK
TITLE = StStarting
//any Transition 
xxS1: S     #Ma.StStarting;
      R     #Ma.Par.OutPulseMat;
      R     #Ma.Par.OutDelayMainValveEnd;
      R     #Ma.Par.OutDelayAirlockEnd;
      L     0;
      T     #Ma.Par.OutDelayTime;
      T     #Ma.Par.OutPulseTime;
      T     #Ma.OutSubState;	//[5.0]
      JU    OUT;
//=== Logic
// Condition for StStopping
S1:   AN    #tmpEnable;
      O     #tmpFaultStop;
      O;
      A     #tmpStoppedMan;
      A     #Ma.InManual;
      R     #Ma.StStarting;
      JC    xxS3;	//--> StStopping
// Condition for StStarted
      A     #Ma.Par.OutDelayMainValveEnd;
      AN    #Ma.Par.ParWithMainValve;
      O     #MainValve.StHN;
      R     #Ma.StStarting;
      JC    xxS2;	//-->StStarted
//Delay main valve
      L     #Ma.Par.ParDelayMain;
      L     #Ma.Par.OutDelayTime;
      <=I;
      O     #MainValve.StHN;
      =     #Ma.Par.OutDelayMainValveEnd;
      AN    "GCS7_Gr_OutTick200ms";	//Gr.OutTick200ms
      O     #Ma.Par.OutDelayMainValveEnd;
      JC    S1J2;
      +     2;
      T     #Ma.Par.OutDelayTime;
S1J2: JU    OUT;
NETWORK
TITLE = StStarted
//any Transition 
xxS2: S     #Ma.StStarted;
      R     #Ma.Par.OutDelayAirlockEnd;
      S     #Ma.Par.OutDelayMainValveEnd;
      L     0;
      T     #Ma.Par.OutDelayTime;
//=== Logic
S2:   L     #Ma.Par.ParDelayAirlock;
      L     #Ma.Par.OutDelayTime;
      <=I;
      =     #Ma.Par.OutDelayAirlockEnd;
// Condition for StFeeding
      A     #Airlock.StStartedFwd;
      A     #Ma.Par.OutDelayAirlockEnd;
      R     #Ma.StStarted;
      JC    xxS6;	//-->StFeeding
// Condition for Clearing
      AN    #tmpEnable;
      O     #tmpClearing;
      O     #tmpFaultStop;
      AN    #Airlock.StStartedFwd;
      O;
      AN    #MainValve.StHN;
      A     #Ma.Par.ParWithMainValve;
      R     #Ma.StStarted;
      JC    xxS5;	//--> StClearing
//Delay Airlock
      AN    "GCS7_Gr_OutTick200ms";	//Gr.OutTick200ms
      O     #Ma.Par.OutDelayAirlockEnd;
      JC    OUT;
      +     2;
      T     #Ma.Par.OutDelayTime;
      JU    OUT;
NETWORK
TITLE = StFeeding
//any Transition 
xxS6: S     #Ma.StFeeding;
      S     #Ma.OutLoaded;
//=== Logic
// Condition for Started
S6:   AN    #Airlock.StStartedFwd;
      R     #Ma.StFeeding;
      JC    xxS2;	//--> StStarted
      JU    OUT;
NETWORK
TITLE = StStopping
//any Transition 
xxS3: S     #Ma.StStopping;
      L     0;
      T     #Ma.Par.OutDelayTime;
      T     #Ma.OutSubState;	//[5.0]
//=== Logic
S3:   L     #Ma.Par.OutDelayTime;
      AN    "GCS7_Gr_OutTick200ms";	//Gr.OutTick200ms
      JC    S3J1;
      +     2;
      T     #Ma.Par.OutDelayTime;
// Condition for StStopped
S3J1: L     #Ma.Par.ParDelayClosing;
      >=I;
      =     #tmpClosingDelayEnd;
      A     #tmpStoppedMan;
      O     #Ma.InManual;
      R     #Ma.StStopping;
      JC    xxS0;	//--> StStopped
      JU    OUT;
NETWORK
TITLE = StClearing
//VV= AirVesselValve
//MV= MatValve
//AV= AirValve
//BV= BypassValve
//
//OutSubState:                            Step          VV    MV    AV    BV 
//     1= ClearingTime Pulsing :                   0     0/1   1/0   0
//     2= AirVesselBlowUp                 1..n     1     0     0     0
//     3= AirVesselPulseOn                1        1     1     0     0
//     4= AirVesselPulseOff               1        0     1     0     0
//     5= AirVesselClearingProduct        1..n     1     1     0     0
//     6= AirVesselClearingBypassProduct  n        1     0     1     0 
//     7= ClearingBoth                    n        1     1     1     0 
//     8= ClearingBypassMain              n+1      0     1     1     1            
//     9= Cleared                         n+1
//
      NOP   0;
//any Transition 
xxS5: S     #Ma.StClearing;
      L     0;
      T     #Ma.Par.OutClearingTime;
      T     #Ma.OutCntClearingCycles;
      T     #Ma.OutCntClearingPulse;
      L     1;
      T     #Ma.OutSubState;
//=== Logic
S5:   NOP   0;
      SET;
      R     #tmpCleared;
//Clearing Time
      AN    "GCS7_Gr_OutTick200ms";	//Gr.OutTick200ms
      JC    S5J0;
      L     #Ma.Par.OutClearingTime;
      +     2;
      T     #Ma.Par.OutClearingTime;
      L     #Ma.Par.OutClearingTimeSubstate;
      +     2;
      T     #Ma.Par.OutClearingTimeSubstate;
S5J0: NOP   0;
//=================================
//OutSubState=1  : Clearing Time    
//=================================
      L     #Ma.OutSubState;
      L     1;
      ==I;
      JCN   C1J0;
      R     #Ma.Par.OutEnableClearingValve;
      R     #Ma.Par.OutEnableBypassValve;
      A     #Ma.Par.OutPulseMat;
      =     #Ma.Par.OutEnableMatValve;
      AN    #Ma.Par.OutPulseMat;
      =     #Ma.Par.OutEnableAirValve;
// ----
      L     #Ma.Par.ParClearingPulsing;
      L     #Ma.Par.OutClearingTime;
      <=I;
      JCN   C1J0;
//Transiton SubState ClearingBoth   
      L     #Ma.InClearingCycles;
      L     0;
      ==I;
      ON    #Ma.Par.ParWithClearingValve;
      JC    CxT7;	//--> SubState: ClearingBoth
//Transiton SubState AirVesselBlowUp   
      L     0;
      T     #Ma.OutCntClearingCycles;
CxT2: L     2;
      T     #Ma.OutSubState;	//--> AirVesselBlowUp
      L     0;
      T     #Ma.Par.OutClearingTimeSubstate;
      T     #Ma.OutCntClearingPulse;
      L     #Ma.OutCntClearingCycles;
      +     1;
      T     #Ma.OutCntClearingCycles;
C1J0: NOP   0;
//===================================
//OutSubState=2  : AirVesselBlowUp
//===================================
      L     #Ma.OutSubState;
      L     2;
      ==I;
      JCN   C2J0;
      S     #Ma.Par.OutEnableClearingValve;
      R     #Ma.Par.OutEnableMatValve;
      R     #Ma.Par.OutEnableAirValve;
      R     #Ma.Par.OutEnableBypassValve;
      AN    #Pressure.InpMax;
      JC    C2J0;
      L     0;
      T     #Ma.OutCntClearingPulse;
//Condition  Step AirVesselPulseOn
      L     #Ma.OutCntClearingCycles;
      L     1;
      ==I;
      JC    CxT3;	//--> SubState AirVesselPulseOn
      L     #Ma.OutCntClearingCycles;
      L     #Ma.InClearingCycles;
      >=I;
      JC    CxT6;	//--> SubState AirVesselClearingBypassProduct    
      JU    CxT5;	//--> SubState AirVesselClearingProduct
//Transition Step     AirVesselPulseOn
CxT3: L     3;	//AirVesselPulseOn
      T     #Ma.OutSubState;
      L     0;
      T     #Ma.Par.OutClearingTimeSubstate;
      L     #Ma.OutCntClearingPulse;
      +     1;
      T     #Ma.OutCntClearingPulse;
      JU    C2J0;
//Transition to SubState AirVesselClearingBypassProduct    
CxT6: L     6;	//          AirVesselClearingBypassProduct  
      T     #Ma.OutSubState;
      L     0;
      T     #Ma.Par.OutClearingTimeSubstate;
      JU    C2J0;
C2J0: NOP   0;
//===================================
//OutSubState=3  = AirVesselPulseOn:
//===================================
      L     #Ma.OutSubState;
      L     3;
      ==I;
      JCN   C3J0;
      S     #Ma.Par.OutEnableClearingValve;
      S     #Ma.Par.OutEnableMatValve;
      R     #Ma.Par.OutEnableAirValve;
      R     #Ma.Par.OutEnableBypassValve;
// ----
      L     #Ma.Par.OutClearingTimeSubstate;
      L     #Ma.Par.ParClearingValvePulseOn;
      <=I;
      JC    C3J0;
CxT4: L     4;	//AirVesselPulseOff
      T     #Ma.OutSubState;
      L     0;
      T     #Ma.Par.OutClearingTimeSubstate;
C3J0: NOP   0;
//===================================
//OutSubState=4  = AirVesselPulseOff:
//===================================
      L     #Ma.OutSubState;
      L     4;
      ==I;
      JCN   C4J0;
      R     #Ma.Par.OutEnableClearingValve;
      S     #Ma.Par.OutEnableMatValve;
      R     #Ma.Par.OutEnableAirValve;
      R     #Ma.Par.OutEnableBypassValve;
//----
      L     #Ma.Par.OutClearingTimeSubstate;
      L     #Ma.Par.ParClearingValvePulseOff;
      <=I;
      JC    C4J0;
      L     #Ma.OutCntClearingPulse;
      L     #Ma.InClearingPulses;
      <I;
      JC    CxT3;	//-->AirVesselPulseOn
//--Transition Substate AirVesselClearing ---
CxT5: L     0;
      T     #Ma.Par.OutClearingTimeSubstate;
      L     5;
      T     #Ma.OutSubState;	//-->AirVesselClearing
C4J0: NOP   0;
//===================================
//OutSubState=5  = AirVesselClearingProduct:
//===================================
      L     #Ma.OutSubState;
      L     5;
      ==I;
      JCN   C5J0;
      S     #Ma.Par.OutEnableClearingValve;
      S     #Ma.Par.OutEnableMatValve;
      R     #Ma.Par.OutEnableAirValve;
      R     #Ma.Par.OutEnableBypassValve;
// ----
      L     #Ma.Par.OutClearingTimeSubstate;
      L     #Ma.Par.ParClearing1stCycle;
      >=I;
      A(;
      L     #Ma.OutCntClearingCycles;
      L     1;
      ==I;
      );
      JC    C5Tx;	//--> Next Step
      L     #Ma.Par.OutClearingTimeSubstate;
      L     #Ma.Par.ParClearing2ndCycle;
      >=I;
      A(;
      L     #Ma.OutCntClearingCycles;
      L     1;
      <>I;
      );
      JC    C5Tx;	//--> Next Step
//Transition SubState AirVesselPulseOff
      L     #Ma.Par.OutClearingTimeSubstate;
      L     #Ma.Par.ParClearingValvePulseOn;
      >I;
      A     #Pressure.InpMax;
      JC    CxT4;
      JU    C5J0;
C5Tx: L     #Ma.OutCntClearingCycles;
      L     #Ma.InClearingCycles;
      <I;
      JC    CxT2;	//-->SubState AirVesselBlowUp
      T     #Ma.OutCntClearingCycles;
C5J0: NOP   0;
//===================================
//OutSubState=6  = AirVesselClearingBypassProduct 
//===================================
      L     #Ma.OutSubState;
      L     6;
      ==I;
      JCN   C6J0;
      S     #Ma.Par.OutEnableClearingValve;
      R     #Ma.Par.OutEnableMatValve;
      S     #Ma.Par.OutEnableAirValve;
      R     #Ma.Par.OutEnableBypassValve;
// ----
      L     #Ma.Par.OutClearingTimeSubstate;
      L     #Ma.Par.ParClearingBypassAirlock;
      >=I;
      JCN   C6J0;
CxT7: L     0;
      T     #Ma.Par.OutClearingTimeSubstate;
      L     7;
      T     #Ma.OutSubState;	//-->ClearingBoth
C6J0: NOP   0;
//===================================
//OutSubState=7  = ClearingBoth:
//===================================
      L     #Ma.OutSubState;
      L     7;
      ==I;
      JCN   C7J0;
      S     #Ma.Par.OutEnableClearingValve;
      S     #Ma.Par.OutEnableMatValve;
      S     #Ma.Par.OutEnableAirValve;
      R     #Ma.Par.OutEnableBypassValve;
// ----
      L     #Ma.Par.OutClearingTimeSubstate;
      L     #Ma.Par.ParClearingBoth;
      >=I;
      JCN   C7J0;
      L     0;
      T     #Ma.Par.OutClearingTimeSubstate;
      L     8;
      T     #Ma.OutSubState;	//-->AirVesselClearingDone
C7J0: NOP   0;
//------------------------------
//OutSubState=8  = ClearingWithBypass:
//------------------------------
      L     #Ma.OutSubState;
      L     8;
      ==I;
      JCN   C8J0;
      R     #Ma.Par.OutEnableClearingValve;
      S     #Ma.Par.OutEnableMatValve;
      S     #Ma.Par.OutEnableAirValve;
      S     #Ma.Par.OutEnableBypassValve;
// ----
      L     #Ma.Par.OutClearingTimeSubstate;
      L     #Ma.Par.ParClearingBypass;
      >=I;
      O     #Ma.InNotClearingBypass;
      JCN   C8J0;
      R     #Ma.OutLoaded;
      L     0;
      T     #Ma.Par.OutClearingTimeSubstate;
      L     9;
      T     #Ma.OutSubState;	//-->Cleared
C8J0: NOP   0;
//------------------------------
//OutSubState=9  = Cleared:
//------------------------------
      L     #Ma.OutSubState;
      L     9;
      ==I;
      JCN   C9J0;
      R     #Ma.Par.OutEnableClearingValve;
      S     #Ma.Par.OutEnableMatValve;
      S     #Ma.Par.OutEnableAirValve;
      R     #Ma.Par.OutEnableBypassValve;
      L     #Ma.Par.OutClearingTimeSubstate;
      L     4;
      >=I;
      =     #tmpCleared;
C9J0: NOP   0;
//------------------------------
// Condition for StStopping
      AN    #Ma.InManual;
      AN    #Ma.InEnable;
      O     #tmpCleared;
      O     #tmpFaultValve;
      O     #Pressure.StFault;	//[5.0]
      O;
      AN    #MainValve.StHN;
      A     #Ma.Par.ParWithMainValve;
      O;
      A     #Ma.InManual;
      AN    #Ma.OutManOpenAll;
      R     #Ma.StClearing;
      JC    xxS3;	//--> StStopping
// Condition for Starting
      A     #tmpEnable;
      AN    #tmpClearing;
      AN    #tmpFaultStop;
      AN    #Ma.InManual;
      R     #Ma.StClearing;
      JC    xxS1;	//--> StStarting
      JU    OUT;
NETWORK
TITLE = State Code
// State           StCode
// ----------------------
// StFault            32
// StStopped          1
// StStarting         2
// StStarted          3
// StFeeding          4
// StClearing         5
// StStopping         7
OUT:  A     #Ma.OutFault;
      L     32;	//Code=Fault
      JC    Code;
      A     #Ma.StStopped;
      L     1;	//Code=Stopped
      JC    Code;
      L     2;	//Code=Starting
      A     #Ma.StStarting;
      JC    Code;
      L     3;	//Code=Started
      A     #Ma.StStarted;
      JC    Code;
      L     4;	//Code=Feeding
      A     #Ma.StFeeding;
      JC    Code;
      L     5;	//Code=Clearing
      A     #Ma.StClearing;
      JC    Code;
      L     7;	//Code=Stopping
Code: L     #Ma.StCode;	// Old state code
      TAK;
      T     #Ma.StCode;	// Save state code
      <>I;
      L     3;
      CC    "SYS_CBitCtrl";	//Set change bit
NETWORK
TITLE = General
      A     #Ma.CmdFaultReset;
      S     #Airlock.CmdFaultReset;
      S     #MainValve.CmdFaultReset;
      S     #MatValve.CmdFaultReset;
      S     #AirValve.CmdFaultReset;
      S     #BypassValve.CmdFaultReset;
      S     #HL.CmdFaultReset;
      S     #SpeedMon.CmdFaultReset;
      S     #Pressure.CmdFaultReset;
      S     #ClearingValve.CmdFaultReset;	//[5.0]
//===  With refill level====
// Pulsing valve
      L     #Ma.Par.OutPulseTime;
      AN    "GCS7_Gr_OutTick200ms";	//Gr.OutTick200ms
      JC    AlJ0;
      +     2;
      T     #Ma.Par.OutPulseTime;
AlJ0: A     #Ma.Par.OutPulseMat;
      JC    ALTC;
      L     #Ma.Par.ParPulseAirTime;
      L     #Ma.Par.OutPulseTime;
      <=I;
      A(;
      ON    #Airlock.StStartedFwd;
      ON    #Ma.Par.ParWithHL;
      );
      O(;
      A     #HL.StCtoTrue;
      O     #HL.StTrue;
      A     #Ma.Par.ParWithHL;
      );
      O;
      A     #Ma.InManual;
      AN    #Ma.OutManPulsing;
      S     #Ma.Par.OutPulseMat;
      JC    AlJ1;
      JU    AlJ3;
AlJ1: L     0;
      T     #Ma.Par.OutPulseTime;
      JU    AlJ3;
ALTC: L     #Ma.Par.ParPulseMatTime;
      L     #Ma.Par.OutPulseTime;
      <=I;
      R     #Ma.Par.OutPulseMat;
      JC    AlJ1;
NETWORK
TITLE = Automatic mode
AlJ3: NOP   0;
      A     #Ma.InManual;
      JC    maJ0;
//Run airlock 
      A     #Ma.StStarted;
      A     #Ma.Par.OutDelayAirlockEnd;
      O     #Ma.StFeeding;
      A     #Ma.InAirOk;
      AN    #Ma.OutFault;
      AN    #Pressure.StCtoOverP;
      AN    #Pressure.StOverP;
      AN    #Pressure.StFault;
      A     #tmpEnable;
      AN    #Ma.InDisableAirlock;
      AN    #Ma.InClearing;
      =     #Airlock.InEnableFwd;
//Pulse-Phase
      A     #Ma.Par.ParWithMatValve;
      AN    #Ma.Par.ParWithAirValve;
      O     #Ma.Par.OutPulseMat;
      =     #tmpReadyConveying;
//Main Valve 
      A     #Ma.Par.OutDelayMainValveEnd;
      S     #MainValve.InEnableHN;
      A     #Ma.StStopped;
      O     #Ma.StStopping;
      R     #MainValve.InEnableHN;
//Air Valve
      A     #Ma.Par.OutEnableAirValve;	//[5.0]
      A     #Ma.StClearing;
      O;
      AN    #Ma.Par.OutPulseMat;
      AN    #Ma.StClearing;
      AN    #Ma.StStopped;
      =     #Ma.Par.OutEnableAirValve;	//[5.0]
      A     #Ma.Par.OutEnableAirValve;	//[5.0]
      S     #AirValve.InEnableHN;
      A     #tmpReadyConveying;
      A     #MatValve.StHN;
      AN    #Ma.Par.OutEnableAirValve;	//[5.0]
      O     #Ma.StStopped;
      O;
      A     #Ma.StStopping;
      A     #tmpClosingDelayEnd;
      O;	//[5.0]
      A     #Ma.Par.OutEnableClearingValve;	//[5.0]
      A     #ClearingValve.StHN;	//[5.0]
      AN    #Ma.Par.OutEnableAirValve;	//[5.0]
      R     #AirValve.InEnableHN;
//Mat Valve
      A     #Ma.Par.OutEnableMatValve;	//[5.0]
      A     #Ma.StClearing;
      O;
      A     #tmpReadyConveying;
      AN    #Ma.StClearing;
      AN    #Ma.StStopped;
      =     #Ma.Par.OutEnableMatValve;	//[5.0]
      A     #Ma.Par.OutEnableMatValve;	//[5.0]
      S     #MatValve.InEnableHN;
//[5.0]     UN    #Ma.Par.OutPulseMat
      A     #AirValve.StHN;
      AN    #Ma.Par.OutEnableMatValve;	//[5.0]
      O     #Ma.StStopped;
      O;
      A     #Ma.StStopping;
      A     #tmpClosingDelayEnd;
      O;
      A     #Ma.Par.OutEnableClearingValve;	//[5.0]
      AN    #Ma.Par.OutEnableMatValve;	//[5.0]
      A     #ClearingValve.StHN;	//[5.0]
      R     #MatValve.InEnableHN;
//Bypass valve 
      AN    #Ma.StClearing;	//[5.0]
      R     #Ma.Par.OutEnableBypassValve;	//[5.0]
      A     #Ma.Par.OutEnableBypassValve;
      S     #BypassValve.InEnableHN;
      AN    #Ma.Par.OutEnableBypassValve;
      R     #BypassValve.InEnableHN;
//ClearingValve [5.0]
      AN    #Ma.StClearing;	//[5.0]
      R     #Ma.Par.OutEnableClearingValve;	//[5.0]
      A     #Ma.Par.OutEnableClearingValve;	//[5.0]
      S     #ClearingValve.InEnableHN;	//[5.0]
      AN    #Ma.Par.OutEnableClearingValve;	//[5.0]
      O     #Pressure.StFault;	//[5.0]
      R     #ClearingValve.InEnableHN;	//[5.0]
NETWORK
TITLE = Manual mode
maJ0: AN    #Ma.InManual;
      JC    AlEn;
//--- Pulsing mode ------------
      A     #Ma.CmdPulsingOnOff;
      A     #Ma.OutManPulsing;
      R     #Ma.OutManPulsing;
      S     #Ma.Par.OutEnableMan;
      JC    maJ1;
      A     #Ma.CmdPulsingOnOff;
      S     #Ma.OutManPulsing;
      R     #Ma.Par.OutEnableMan;
      R     #Ma.OutManOpenAll;
//-- Airlock ------------------- 
maJ1: A     #Ma.CmdAirlockOnOff;
      A     #Airlock.StStopped;
      S     #Airlock.InEnableFwd;
      S     #Airlock.CmdNext;
// 
      A     #Ma.CmdAirlockOnOff;
      AN    #Airlock.StStopped;
      O;
      AN    #MainValve.StHN;
      A     #Ma.Par.ParWithMainValve;
      O     #Ma.OutFault;
      O     #Pressure.StCtoOverP;
      O     #Pressure.StOverP;
      O     #Pressure.StFault;
      O     #Ma.CmdOff;
      O     #Ma.InDisableAirlock;
      R     #Airlock.InEnableFwd;
//---- Main Valve -------------- 
      A     #Ma.CmdMainOnOff;
      R     #Ma.OutManOpenAll;
      A     #Ma.CmdMainOnOff;
      A     #MainValve.StLN;
      S     #MainValve.InEnableHN;
      A     #Ma.CmdMainOnOff;
      AN    #MainValve.StLN;
      O     #Ma.CmdOff;
      R     #MainValve.InEnableHN;
//--- MatValve - AirValve --------- 
      A     #Ma.Par.OutPulseMat;
      A     #Ma.OutManPulsing;
      O;
      AN    #Ma.OutManPulsing;
      A     #Ma.Par.OutEnableMan;
      S     #MatValve.InEnableHN;
      =     #tmpVKE;
      A     #tmpVKE;
      A     #MatValve.StHN;
      R     #AirValve.InEnableHN;
// 
      AN    #Ma.Par.OutPulseMat;
      A     #Ma.OutManPulsing;
      AN    #Ma.OutManOpenAll;
      S     #AirValve.InEnableHN;
      =     #tmpVKE;
      A     #tmpVKE;
      A     #AirValve.StHN;
      R     #MatValve.InEnableHN;
//--BypassV--- 
      A     #Ma.OutManPulsing;
      R     #BypassValve.InEnableHN;
//--- Open All--------------------     
      A     #Ma.CmdOpenAll;
      S     #Ma.OutManOpenAll;
      R     #Ma.OutManPulsing;
      A     #Ma.OutManOpenAll;
      S     #BypassValve.InEnableHN;
      S     #MatValve.InEnableHN;
      S     #AirValve.InEnableHN;
      S     #MainValve.InEnableHN;
//--- Off ------------------------ 
      A     #Ma.CmdOff;
      R     #Ma.OutManOpenAll;
      R     #Ma.OutManPulsing;
      R     #Ma.Par.OutEnableMan;
      R     #MainValve.InEnableHN;
      R     #BypassValve.InEnableHN;
      R     #MatValve.InEnableHN;
      R     #AirValve.InEnableHN;
// 
NETWORK
TITLE = Global End
AlEn: AN    #BypassValve.InEnableHN;
      =     #BypassValve.InEnableLN;
      AN    #MatValve.InEnableHN;
      =     #MatValve.InEnableLN;
      AN    #AirValve.InEnableHN;
      =     #AirValve.InEnableLN;
      AN    #MainValve.InEnableHN;
      =     #MainValve.InEnableLN;
      AN    #ClearingValve.InEnableHN;	//[5.0]
      =     #ClearingValve.InEnableLN;	//[5.0]
//Init Pressure     //[5.0]
//Transition StCtoOverP --> StNormalP      
      A     #Pressure.StCtoOverP;	//[5.0]
      A     #ClearingValve.StHN;	//[5.0]
      AN    #Pressure.InpMax;	//[5.0]
      AN    #Pressure.InpMin;	//[5.0]
      S     #Pressure.StNormalP;	//[5.0]
      R     #Pressure.StCtoOverP;	//[5.0]
//Next
      A     #Ma.CmdNext;
      O     #Ma.InManual;
      S     #Airlock.CmdNext;
      SET;
      S     #BypassValve.CmdNext;
      S     #MatValve.CmdNext;
      S     #AirValve.CmdNext;
      S     #MainValve.CmdNext;
      S     #ClearingValve.CmdNext;	//[5.0]
//---Clear all commands
      CLR;
      =     #Ma.CmdMainOnOff;
      =     #Ma.CmdOff;
      =     #Ma.CmdNext;
      =     #Ma.CmdFaultReset;
      =     #Ma.CmdAirlockOnOff;
      =     #Ma.CmdOpenAll;
      =     #Ma.CmdPulsingOnOff;
// 
END_FUNCTION_BLOCK

